# B&R Automation Studio project DuctLines (part 5)

#### Server.st - Cyclic code
```iecst
(********************************************************************
 ********************************************************************
 * Program: Server
 * File: Server.st
 * Created: May, 2018
 ********************************************************************
 * Implementation of program Server
 ********************************************************************)

PROGRAM _CYCLIC

	CASE Server.sStep OF

		0:  (* Open Ethernet Interface *)
			Server.TcpOpen_0.enable := 1;
			Server.TcpOpen_0.pIfAddr := 0;  (* Listen on all TCP/IP Interfaces*)
			Server.TcpOpen_0.port := 12000;  (* Port to listen*)
			Server.TcpOpen_0.options := 0;
			Server.TcpOpen_0;  (* Call the Function*)

			IF Server.TcpOpen_0.status = 0 THEN  (* TcpOpen successfull*)
				Server.sStep := 5;
			ELSIF Server.TcpOpen_0.status = ERR_FUB_BUSY THEN  (* TcpOpen not finished -> redo *)
				(* Busy *)
			ELSE  (* Goto Error Step *)
				Server.recv_timeout := 0;
				Server.sStep := 100;
			END_IF

		5:
			Server.linger_opt.lLinger := 0; (* linger Time = 0 *)
			Server.linger_opt.lOnOff := 1; (* linger Option ON *)
			Server.TcpIoctl_0.enable := 1;
			Server.TcpIoctl_0.ident := Server.TcpOpen_0.ident; (* Connection Ident from AsTCP.TCP_Open *)
			Server.TcpIoctl_0.ioctl := tcpSO_LINGER_SET; (* Set Linger Options *)
			Server.TcpIoctl_0.pData := ADR(Server.linger_opt);
			Server.TcpIoctl_0.datalen := SIZEOF(Server.linger_opt);
			Server.TcpIoctl_0;

			IF Server.TcpIoctl_0.status = 0 THEN  (* TcpIoctl successfull *)
				Server.sStep := 10;
			ELSIF Server.TcpIoctl_0.status = ERR_FUB_BUSY THEN  (* TcpIoctl not finished -> redo *)
				(* Busy *)
			ELSE  (* Goto Error Step *)
				Server.recv_timeout := 0;
				Server.sStep := 100;
			END_IF

		10: (* Wait for Client Connection *)
			Server.TcpServer_0.enable := 1;
			Server.TcpServer_0.ident := Server.TcpOpen_0.ident;  (* Connection Ident from AsTCP.TCP_Open *)
			Server.TcpServer_0.backlog := 1;  (* Number of clients waiting simultaneously for a connection*)
			Server.TcpServer_0.pIpAddr := ADR(Server.client_address);  (* Where to write the client IP-Address*)
			Server.TcpServer_0;  (* Call the Function*)

			IF Server.TcpServer_0.status = 0 THEN  (* Status = 0 if an client connects to server *)
				Server.sStep := 15;
			ELSIF Server.TcpServer_0.status = ERR_FUB_BUSY THEN  (* TcpServer not finished -> redo *)
				(* Busy *)
			ELSE  (* Goto Error Step *)
				Server.recv_timeout := 0;
				Server.sStep := 100;
			END_IF

		15:
			Server.TcpIoctl_0.enable := 1;
			Server.TcpIoctl_0.ident := Server.TcpServer_0.identclnt; (* Connection Ident from AsTCP.TCP_Server *)
			Server.TcpIoctl_0.ioctl := tcpSO_LINGER_SET;  (* Set Linger Options *)
			Server.TcpIoctl_0.pData := ADR(Server.linger_opt);
			Server.TcpIoctl_0.datalen := SIZEOF(Server.linger_opt);
			Server.TcpIoctl_0;

			IF Server.TcpIoctl_0.status = 0 THEN  (* TcpIoctl successfull *)
				Server.sStep := 20;
			ELSIF Server.TcpIoctl_0.status = ERR_FUB_BUSY THEN  (* TcpIoctl not finished -> redo *)
				(* Busy *)
			ELSE  (* Goto Error Step *)
				Server.recv_timeout := 0;
				Server.sStep := 100;
			END_IF

		20: (* Wait for Data *)
			Server.TcpRecv_0.enable := 1;
			Server.TcpRecv_0.ident := Server.TcpServer_0.identclnt;  (* Client Ident from AsTCP.TCP_Server *)
			Server.TcpRecv_0.pData	:= ADR(Server.data_buffer);  (* Where to store the incoming data *)
			Server.TcpRecv_0.datamax := SIZEOF(Server.data_buffer);  (* Length of data buffer *)
			Server.TcpRecv_0.flags := 0;
			Server.TcpRecv_0;  (* Call the Function*)

			IF Server.TcpRecv_0.status = 0 THEN
				(* This gets Server.sStep out of here when the PC program stop executing*)
				Server.recv_timeout := Server.recv_timeout + 1;
				IF Server.recv_timeout > 250 THEN
					Server.sStep := 40;
					Server.recv_timeout := 0;
				END_IF
			ELSIF Server.TcpRecv_0.status = tcpERR_NO_DATA THEN
				(*This criteria isn't true when the PC program isn't executing*)
				Server.recv_timeout := Server.recv_timeout + 1;
				IF Server.recv_timeout > 500 THEN
					Server.sStep := 40;
					Server.recv_timeout := 0;
				END_IF
			ELSIF Server.TcpRecv_0.status = ERR_FUB_BUSY THEN

			ELSIF Server.TcpRecv_0.status = tcpERR_NOT_CONNECTED THEN
				(* This doesn't appear to work.*)
				Server.sStep := 40;
			ELSE
				Server.recv_timeout := 0;
				Server.sStep := 100;
			END_IF

			LastByte := Server.TcpRecv_0.recvlen - 3;
			IF Server.data_buffer[LastByte] = 13 THEN
				(*Receive Transmission Complete, Parse Data*)
				Server.recv_timeout := 0;
				Server.data_buffer[LastByte] := 0;
				HandleIndex := 0;
				UpperLimit := LastByte; (* Parsing Loop Will Run To Here *)
				TrueString := 'True';
				Server.sStep := 25;
				(*Server.sStep := 90;*)
			END_IF
		25: (* Parse Out Values *)
			REPEAT
				(* Get The Tag Handle *)
				CommaPosition1 := HandleIndex;
				WHILE Server.data_buffer[CommaPosition1] <> 44 DO
					CommaPosition1 := CommaPosition1 + 1;
				END_WHILE;
				SLength := CommaPosition1 - HandleIndex;
				nxt_adr := memmove(ADR(HandleStringA), ADR(Server.data_buffer[HandleIndex]), SLength);
				HandleStringB := LEFT(HandleStringA, UDINT_TO_INT(SLength));
				TagHandle := atoi(ADR(HandleStringB));
				HandleIndex := CommaPosition1 + 1;

				(* Get The String Containing The Value *)
				CommaPosition1 := HandleIndex;
				WHILE Server.data_buffer[CommaPosition1] <> 44 DO
					CommaPosition1 := CommaPosition1 + 1;
				END_WHILE;
				SLength := CommaPosition1 - HandleIndex;
				nxt_adr := memmove(ADR(ValueStringA), ADR(Server.data_buffer[HandleIndex]), SLength);
				ValueStringB := LEFT(ValueStringA, UDINT_TO_INT(SLength));
				HandleIndex := CommaPosition1 + 1;
				CASE TagHandle OF
					0:
						RunJob := atoi(ADR(ValueStringB));
					1:
						IF strcmp(ADR(TrueString), ADR(ValueStringB)) = 0 THEN
							RunJobClick := TRUE;
						ELSE
							RunJobClick := FALSE;
						END_IF;
					2:
						NewRunJob := atoi(ADR(ValueStringB));
					3:
						IF strcmp(ADR(TrueString), ADR(ValueStringB)) = 0 THEN
							StartSignal := TRUE;
						ELSE
							StartSignal := FALSE;
						END_IF;
					4..9:
						ShearTable[TagHandle - 4] := atof(ADR(ValueStringB));
					10..15:
						LTNotchTable[TagHandle - 10] := atof(ADR(ValueStringB));
					16..21:
						VNotchTable[TagHandle - 16] := atof(ADR(ValueStringB));
					22..39:
						LeftHoleTable[TagHandle - 22] := atof(ADR(ValueStringB));
					40..57:
						CenterHoleTable[TagHandle - 40] := atof(ADR(ValueStringB));
					58..75:
						RightHoleTable[TagHandle - 58] := atof(ADR(ValueStringB));
					76:
						ShearHits := atoi(ADR(ValueStringB));
					77:
						LTNotchHits := atoi(ADR(ValueStringB));
					78:
						VNotchHits := atoi(ADR(ValueStringB));
					79:
						LeftHoleHits := atoi(ADR(ValueStringB));
					80:
						CenterHoleHits := atoi(ADR(ValueStringB));
					81:
						RightHoleHits := atoi(ADR(ValueStringB));
					82:
						IF strcmp(ADR(TrueString), ADR(ValueStringB)) = 0 THEN
							SealantRequired := TRUE;
						ELSE
							SealantRequired := FALSE;
						END_IF;
					83:
						IF strcmp(ADR(TrueString), ADR(ValueStringB)) = 0 THEN
							CropCut := TRUE;
						ELSE
							CropCut := FALSE;
						END_IF;
					84:
						WarningDelay1 := DINT_TO_TIME(atoi(ADR(ValueStringB)));
					85:
						PartsMade := atoi(ADR(ValueStringB));
					86:
						MetalDesired := atof(ADR(ValueStringB));
					87:
						MetalActual := atof(ADR(ValueStringB));
					88:
						IF strcmp(ADR(TrueString), ADR(ValueStringB)) = 0 THEN
							InCycle := TRUE;
						ELSE
							InCycle := FALSE;
						END_IF;
					89:
						PercentSpeed1 := atoi(ADR(ValueStringB));
					90:
						CropPercent1 := atoi(ADR(ValueStringB));
					91:
						TotalInches := atof(ADR(ValueStringB));
					92:
						PartLength := atof(ADR(ValueStringB));
					93:
					94:
						IF strcmp(ADR(TrueString), ADR(ValueStringB)) = 0 THEN
							MakeShearTable := TRUE;
						ELSE
							MakeShearTable := FALSE;
						END_IF;
					95:
						IF strcmp(ADR(TrueString), ADR(ValueStringB)) = 0 THEN
							MakeLTTable := TRUE;
						ELSE
							MakeLTTable := FALSE;
						END_IF;
					96:
						IF strcmp(ADR(TrueString), ADR(ValueStringB)) = 0 THEN
							MakeVTable := TRUE;
						ELSE
							MakeVTable := FALSE;
						END_IF;
					97:
						IF strcmp(ADR(TrueString), ADR(ValueStringB)) = 0 THEN
							MakeLHoleTable := TRUE;
						ELSE
							MakeLHoleTable := FALSE;
						END_IF;
					98:
						IF strcmp(ADR(TrueString), ADR(ValueStringB)) = 0 THEN
							MakeCHoleTable := TRUE;
						ELSE
							MakeCHoleTable := FALSE;
						END_IF;
					99:
						IF strcmp(ADR(TrueString), ADR(ValueStringB)) = 0 THEN
							MakeRHoleTable := TRUE;
						ELSE
							MakeRHoleTable := FALSE;
						END_IF;
					100:
						ShearFFlag := atoi(ADR(ValueStringB));
					101:
						NotchFFlag1 := atoi(ADR(ValueStringB));
					102:
						IF strcmp(ADR(TrueString), ADR(ValueStringB)) = 0 THEN
							BatchCancelSignal := TRUE;
						ELSE
							BatchCancelSignal := FALSE;
						END_IF;
					103:
						IF strcmp(ADR(TrueString), ADR(ValueStringB)) = 0 THEN
							RunContinuousSignal := TRUE;
						ELSE
							RunContinuousSignal := FALSE;
						END_IF;
					104:
						ShearJob := atoi(ADR(ValueStringB));
					105:
						LTJob := atoi(ADR(ValueStringB));
					106:
						VJob := atoi(ADR(ValueStringB));
					107:
						LHoleJob := atoi(ADR(ValueStringB));
					108:
					    BackGaugeJogPercent := atoi(ADR(ValueStringB)); (*Iowa Servo Brake Uses This, too*)
					109:
					    RHoleJob := atoi(ADR(ValueStringB)); (* Iowa *)
					    BackGaugeRunPercent := RHoleJob; (* Engel *)
					110:
						ShearDwell := atoi(ADR(ValueStringB));
					111:
						LTDwell := atoi(ADR(ValueStringB));
					112:
						VDwell := atoi(ADR(ValueStringB));
					113:
						LHoleDwell := atoi(ADR(ValueStringB));
					114:
						CHoleDwell := atoi(ADR(ValueStringB));
					115:
						RHoleDwell := atoi(ADR(ValueStringB));
					116:
						GapTime := atoi(ADR(ValueStringB));
					117..134:
						IF strcmp(ADR(TrueString), ADR(ValueStringB)) = 0 THEN
							LeftDiePosition[TagHandle - 117] := TRUE;
						ELSE
							LeftDiePosition[TagHandle - 117] := FALSE;
						END_IF;
					135..152:
						IF strcmp(ADR(TrueString), ADR(ValueStringB)) = 0 THEN
							CenterDiePosition[TagHandle - 135] := TRUE;
						ELSE
							CenterDiePosition[TagHandle - 135] := FALSE;
						END_IF;
					153..170:
						IF strcmp(ADR(TrueString), ADR(ValueStringB)) = 0 THEN
							RightDiePosition[TagHandle - 153] := TRUE;
						ELSE
							RightDiePosition[TagHandle - 153] := FALSE;
						END_IF;
					171:
						LTRemainder := atof(ADR(ValueStringB));
					172:
						VRemainder := atof(ADR(ValueStringB));
					173:
						LHoleRemainder := atof(ADR(ValueStringB));
					174:
						CHoleRemainder := atof(ADR(ValueStringB));
					175:
						RHoleRemainder := atof(ADR(ValueStringB));
					176:
						PercentJogSpeed1 := atoi(ADR(ValueStringB));
					177:
						MetalEncoder := atoi(ADR(ValueStringB));
					178:
						MarkEncoder := atoi(ADR(ValueStringB));
					179:
						PinspotEncoder := atoi(ADR(ValueStringB));
					180:
						BrakeEncoder := atoi(ADR(ValueStringB));
					181:
						IF strcmp(ADR(TrueString), ADR(ValueStringB)) = 0 THEN
							RollDriveEnableButton := TRUE;
						ELSE
							RollDriveEnableButton := FALSE;
						END_IF;
					182:
					(*Lift3DownDwell := STRING_TO_TIME(ValueStringB);*)
					    Lift3DownDwell := DINT_TO_TIME(atoi(ADR(ValueStringB)));
					183:
					(*Lift3UpDwell := STRING_TO_TIME(alueStringB);*)
					    Lift3UpDwell := DINT_TO_TIME(atoi(ADR(ValueStringB)));
					184:
						EngelBrakeModelNumber := atoi(ADR(ValueStringB));
					185:
						IF strcmp(ADR(TrueString), ADR(ValueStringB)) = 0 THEN
							SideDischargeBrake := TRUE;
						ELSE
							SideDischargeBrake := FALSE;
						END_IF;
					186: (* The E1000 PC program turns this on. *)
						IF strcmp(ADR(TrueString), ADR(ValueStringB)) = 0 THEN
							E1000CoilLine := TRUE;
						ELSE
							E1000CoilLine := FALSE;
						END_IF;
					187:
						BrakeEjectTarget := atof(ADR(ValueStringB));
					188..272: (*Obsolete Data*)
					273:
						LatestConnector := DINT_TO_INT(atoi(ADR(ValueStringB)));
					274:
						IF strcmp(ADR(TrueString), ADR(ValueStringB)) = 0 THEN
							WaitToFire1 := TRUE;
						ELSE
							WaitToFire1 := FALSE;
						END_IF;
					275:
						IF strcmp(ADR(TrueString), ADR(ValueStringB)) = 0 THEN
							WaitToFire2 := TRUE;
						ELSE
							WaitToFire2 := FALSE;
						END_IF;
					276:
						IF strcmp(ADR(TrueString), ADR(ValueStringB)) = 0 THEN
							WaitToFire3 := TRUE;
						ELSE
							WaitToFire3 := FALSE;
						END_IF;
					277: (*Obsolete Boolean*)
					278:
						MarkTableDecelDelay := atoi(ADR(ValueStringB));
					279:
						MarkGateUpDwell := atoi(ADR(ValueStringB));
					280:
						MarkPStartDelay := atoi(ADR(ValueStringB));
					281:
						MarkPPauseDwell := atoi(ADR(ValueStringB));
					282:
						MarkPStageTime := atoi(ADR(ValueStringB));
					283:
						MarkPStopDelay := atoi(ADR(ValueStringB));
					284:
						IF strcmp(ADR(TrueString), ADR(ValueStringB)) = 0 THEN
							BeginMarkHoming := TRUE;
						ELSE
							BeginMarkHoming := FALSE;
						END_IF;
					285:
						MarkTarget := atof(ADR(ValueStringB));
					286:
						MarkInPosBand := atoi(ADR(ValueStringB));
					287:
						MarkSlowBand := atoi(ADR(ValueStringB));
					288:
						MarkReference := atof(ADR(ValueStringB));
					289:
						MarkResolution := atof(ADR(ValueStringB));
					290:
						MarkStatus := atoi(ADR(ValueStringB));
					291:
						MarkMinLength := atof(ADR(ValueStringB));
					292:
						MarkDesired := atof(ADR(ValueStringB));
					293:
						MarkActual := atof(ADR(ValueStringB));
					294:
						IF strcmp(ADR(TrueString), ADR(ValueStringB)) = 0 THEN
							ClearLengthCountSignal := TRUE;
						ELSE
							ClearLengthCountSignal := FALSE;
						END_IF;
					295:
						IF strcmp(ADR(TrueString), ADR(ValueStringB)) = 0 THEN
							MarkButtonSignal := TRUE;
						ELSE
							MarkButtonSignal := FALSE;
						END_IF;
					296:
						IF strcmp(ADR(TrueString), ADR(ValueStringB)) = 0 THEN
							MarkSetSignal := TRUE;
						ELSE
							MarkSetSignal := FALSE;
						END_IF;
					297:
						TDCPushSetupDwell := atoi(ADR(ValueStringB));
					298:
						TDCSquareDelay := atoi(ADR(ValueStringB));
					299:
						TDCTablePauseDwell := atoi(ADR(ValueStringB));
					300:
						PinspotResolution := atof(ADR(ValueStringB));
					301:
						PSpotDesired := atof(ADR(ValueStringB));
					302:
						PSpotActual := atof(ADR(ValueStringB));
					303:
						IF strcmp(ADR(TrueString), ADR(ValueStringB)) = 0 THEN
							PinsRequired := TRUE;
						ELSE
							PinsRequired := FALSE;
						END_IF;
					304:
						PinTarget0 := atof(ADR(ValueStringB));
					305:
						PinTarget1 := atof(ADR(ValueStringB));
					306:
						PinTarget2 := atof(ADR(ValueStringB));
					307:
						PinTarget3 := atof(ADR(ValueStringB));
					308:
						PinTarget4 := atof(ADR(ValueStringB));
					309:
						PinTarget5 := atof(ADR(ValueStringB));
					310:
						PinTarget6 := atof(ADR(ValueStringB));
					311:
						PinTarget7 := atof(ADR(ValueStringB));
					312:
						PinTarget8 := atof(ADR(ValueStringB));
					313:
						PinTarget9 := atof(ADR(ValueStringB));
					314:
						PinRepeat0 := atoi(ADR(ValueStringB));
					315:
						PinRepeat1 := atoi(ADR(ValueStringB));
					316:
						PinRepeat2 := atoi(ADR(ValueStringB));
					317:
						PinRepeat3 := atoi(ADR(ValueStringB));
					318:
						PinRepeat4 := atoi(ADR(ValueStringB));
					319:
						PinRepeat5 := atoi(ADR(ValueStringB));
					320:
						PinRepeat6 := atoi(ADR(ValueStringB));
					321:
						PinRepeat7 := atoi(ADR(ValueStringB));
					322:
						PinRepeat8 := atoi(ADR(ValueStringB));
					323:
						PinRepeat9 := atoi(ADR(ValueStringB));
					324:
						PinDriveDwell := atoi(ADR(ValueStringB));
					325:
						PinLoadDwell := atoi(ADR(ValueStringB));
					326:
						PinLoadDelay := atoi(ADR(ValueStringB));
					327:
						IF strcmp(ADR(TrueString), ADR(ValueStringB)) = 0 THEN
							PinspotterSetSignal := TRUE;
						ELSE
							PinspotterSetSignal := FALSE;
						END_IF;
					328:
						IF strcmp(ADR(TrueString), ADR(ValueStringB)) = 0 THEN
							BrakeRefSignal := TRUE;
						ELSE
							BrakeRefSignal := FALSE;
						END_IF;
					329:
						BrakeReference := atof(ADR(ValueStringB));
					330:
						BrakeTarget0 := atof(ADR(ValueStringB));
					331:
						BrakeTarget1 := atof(ADR(ValueStringB));
					332:
						BrakeTarget2 := atof(ADR(ValueStringB));
					333:
						BrakeTarget3 := atof(ADR(ValueStringB));
					334:
						IF strcmp(ADR(TrueString), ADR(ValueStringB)) = 0 THEN
							BrakeRequired := TRUE;
						ELSE
							BrakeRequired := FALSE;
						END_IF;
					335:
						BrakeSlowWindow := atoi(ADR(ValueStringB)); (*Iowa*)
					    CoilLineSlowWindow := BrakeSlowWindow; (*Engel*)
					336:
						BrakeTargetWindow := atoi(ADR(ValueStringB)); (*Iowa*)
					    CoilLineTargetWindow := BrakeTargetWindow; (*Engel*)
					337:
						BrakeDesired := atof(ADR(ValueStringB));
					338:
						BrakeActual := atof(ADR(ValueStringB));
					339:
						BrakeResolution := atof(ADR(ValueStringB));
					340:
						DuctType := atoi(ADR(ValueStringB));
					341:
						BrakeStatus := atoi(ADR(ValueStringB));
					342:
						IF strcmp(ADR(TrueString), ADR(ValueStringB)) = 0 THEN
							PCBrakeSetSignal := TRUE;
						ELSE
							PCBrakeSetSignal := FALSE;
						END_IF;
					343:
						IF strcmp(ADR(TrueString), ADR(ValueStringB)) = 0 THEN
							FBBrakeSetSignal := TRUE;
						ELSE
							FBBrakeSetSignal := FALSE;
						END_IF;
					344:
						IF strcmp(ADR(TrueString), ADR(ValueStringB)) = 0 THEN
							ULineSelected := TRUE;
						ELSE
							ULineSelected := FALSE;
						END_IF;
					345:
						IF strcmp(ADR(TrueString), ADR(ValueStringB)) = 0 THEN
							ZeroCropCut := TRUE;
						ELSE
							ZeroCropCut := FALSE;
						END_IF;
					346:
						IF strcmp(ADR(TrueString), ADR(ValueStringB)) = 0 THEN
							Short2ndLeg := TRUE;
						ELSE
							Short2ndLeg := FALSE;
						END_IF;
					347:
						IF strcmp(ADR(TrueString), ADR(ValueStringB)) = 0 THEN
							HWBrakeWithPLC := TRUE;
						ELSE
							HWBrakeWithPLC := FALSE;
						END_IF;
					348:
						IF strcmp(ADR(TrueString), ADR(ValueStringB)) = 0 THEN
							LBrakeWithPLC := TRUE;
						ELSE
							LBrakeWithPLC := FALSE;
						END_IF;
					349:
						IF strcmp(ADR(TrueString), ADR(ValueStringB)) = 0 THEN
							CycleShear := TRUE;
						ELSE
							CycleShear := FALSE;
						END_IF;
					350:
						IF strcmp(ADR(TrueString), ADR(ValueStringB)) = 0 THEN
							CycleLTDie := TRUE;
						ELSE
							CycleLTDie := FALSE;
						END_IF;
					351:
						IF strcmp(ADR(TrueString), ADR(ValueStringB)) = 0 THEN
							CycleVDie := TRUE;
						ELSE
							CycleVDie := FALSE;
						END_IF;
					352:
						IF strcmp(ADR(TrueString), ADR(ValueStringB)) = 0 THEN
							CycleLDie := TRUE;
						ELSE
							CycleLDie := FALSE;
						END_IF;
					353:
						IF strcmp(ADR(TrueString), ADR(ValueStringB)) = 0 THEN
							CycleCDie := TRUE;
						ELSE
							CycleCDie := FALSE;
						END_IF;
					354:
						IF strcmp(ADR(TrueString), ADR(ValueStringB)) = 0 THEN
							CycleRDie := TRUE;
						ELSE
							CycleRDie := FALSE;
						END_IF;
					355:
						IF strcmp(ADR(TrueString), ADR(ValueStringB)) = 0 THEN
							SpareBool1 := TRUE;
						ELSE
							SpareBool1 := FALSE;
						END_IF;
					356:
						IF strcmp(ADR(TrueString), ADR(ValueStringB)) = 0 THEN
							ShearBrakeLatch := TRUE;
						ELSE
							ShearBrakeLatch := FALSE;
						END_IF;
					357:
						IF strcmp(ADR(TrueString), ADR(ValueStringB)) = 0 THEN
							CycleCustomVDie := TRUE;
						ELSE
							CycleCustomVDie := FALSE;
						END_IF;
					358:
						IF strcmp(ADR(TrueString), ADR(ValueStringB)) = 0 THEN
							CycleCustomLTDie := TRUE;
						ELSE
							CycleCustomLTDie := FALSE;
						END_IF;
					359:
						IF strcmp(ADR(TrueString), ADR(ValueStringB)) = 0 THEN
							SpareBool2 := TRUE;
						ELSE
							SpareBool2 := FALSE;
						END_IF;
					360:
						IF strcmp(ADR(TrueString), ADR(ValueStringB)) = 0 THEN
							SpareBool3 := TRUE;
						ELSE
							SpareBool3 := FALSE;
						END_IF;
					361:
						CustomLTDwell := atoi(ADR(ValueStringB));
					362:
						CustomVDwell := atoi(ADR(ValueStringB));
					363:
						TDCRFPusherStopDelay := atoi(ADR(ValueStringB));
					364:
						GlueApplicatorType := atoi(ADR(ValueStringB));
					365:
						IF strcmp(ADR(TrueString), ADR(ValueStringB)) = 0 THEN
							MakeButtonTable := TRUE;
						ELSE
							MakeButtonTable := FALSE;
						END_IF;
					366:
						IF strcmp(ADR(TrueString), ADR(ValueStringB)) = 0 THEN
							MakeShearBrakeTable := TRUE;
						ELSE
							MakeShearBrakeTable := FALSE;
						END_IF;
					367:
						IF strcmp(ADR(TrueString), ADR(ValueStringB)) = 0 THEN
							MakeCustomLTTable := TRUE;
						ELSE
							MakeCustomLTTable := FALSE;
						END_IF;
					368:
						IF strcmp(ADR(TrueString), ADR(ValueStringB)) = 0 THEN
							MakeCleatTable := TRUE;
						ELSE
							MakeCleatTable := FALSE;
						END_IF;
					369:
						ButtonHits := atoi(ADR(ValueStringB));
					370:
						ShearBrakeHits := atoi(ADR(ValueStringB));
					371:
						CustomLTHits := atoi(ADR(ValueStringB));
					372:
						CleatHits := atoi(ADR(ValueStringB));
					373:
						ButtonJob := atoi(ADR(ValueStringB));
					374:
						ShearBrakeJob := atoi(ADR(ValueStringB));
					375:
						CustomLTJob := atoi(ADR(ValueStringB));
					376:
						CleatJob := atoi(ADR(ValueStringB));
					377:
						ButtonRemainder := atof(ADR(ValueStringB));
					378:
						ShearBrakeRemainder := atof(ADR(ValueStringB));
					379:
						CustomLTRemainder := atof(ADR(ValueStringB));
					380:
						CleatRemainder := atof(ADR(ValueStringB));
					381..386:
						ButtonTable[TagHandle - 381] := atof(ADR(ValueStringB));
					387..392:
						ShearBrakeTable[TagHandle - 387] := atof(ADR(ValueStringB));
					393..398:
						CustomLTTable[TagHandle - 393] := atof(ADR(ValueStringB));
					399..404:
						CleatTable[TagHandle - 399] := atof(ADR(ValueStringB));
					405:
						DieUpDelay := atoi(ADR(ValueStringB));
					406:
						IF strcmp(ADR(TrueString), ADR(ValueStringB)) = 0 THEN
							BrakeAuto := TRUE;
						ELSE
							BrakeAuto := FALSE;
						END_IF;
					407:
						IF strcmp(ADR(TrueString), ADR(ValueStringB)) = 0 THEN
							DuctSelected := TRUE;
						ELSE
							DuctSelected := FALSE;
						END_IF;
					408:
						IF strcmp(ADR(TrueString), ADR(ValueStringB)) = 0 THEN
							EngelEServoOption := TRUE;
						ELSE
							EngelEServoOption := FALSE;
						END_IF;
					409:
						IF strcmp(ADR(TrueString), ADR(ValueStringB)) = 0 THEN
							ConfigureServos := TRUE;
						ELSE
							ConfigureServos := FALSE;
						END_IF;
					410:
						IF strcmp(ADR(TrueString), ADR(ValueStringB)) = 0 THEN
							SpareBool4 := TRUE;
						ELSE
							SpareBool4 := FALSE;
						END_IF;
					411:
						IF strcmp(ADR(TrueString), ADR(ValueStringB)) = 0 THEN
							SpareBool5 := TRUE;
						ELSE
							SpareBool5 := FALSE;
						END_IF;
					412:
						NotchFFlag2 := atoi(ADR(ValueStringB));
					413:
						ITmr1 := atoi(ADR(ValueStringB));
					414:
						ITmr2 := atoi(ADR(ValueStringB));
					415:
						ITmr3 := atoi(ADR(ValueStringB));
					416:
						ITmr4 := atoi(ADR(ValueStringB));
					417:
						ITmr5 := atoi(ADR(ValueStringB));
					418:
						ITmr6 := atoi(ADR(ValueStringB));
					419:
						ITmr7 := atoi(ADR(ValueStringB));
					420:
						ITmr8 := atoi(ADR(ValueStringB));
					421:
						ITmr9 := atoi(ADR(ValueStringB));
					422:
						ITmr10 := atoi(ADR(ValueStringB));
					423:
						ITmr11 := atoi(ADR(ValueStringB));
					424:
						ITmr12 := atoi(ADR(ValueStringB));
					425:
						ITmr13 := atoi(ADR(ValueStringB));
					426:
						IF strcmp(ADR(TrueString), ADR(ValueStringB)) = 0 THEN
							InsulationRequired := TRUE;
						ELSE
							InsulationRequired := FALSE;
						END_IF;
					427:
						IF strcmp(ADR(TrueString), ADR(ValueStringB)) = 0 THEN
							HeartBeat := TRUE;
						ELSE
							HeartBeat := FALSE;
						END_IF;
					428:
						IF strcmp(ADR(TrueString), ADR(ValueStringB)) = 0 THEN
							TDCRunSignal := TRUE;
						ELSE
							TDCRunSignal := FALSE;
						END_IF;
					429:
						IF strcmp(ADR(TrueString), ADR(ValueStringB)) = 0 THEN
							TDCRFMotor := TRUE;
						ELSE
							TDCRFMotor := FALSE;
						END_IF;
					430:
						IF strcmp(ADR(TrueString), ADR(ValueStringB)) = 0 THEN
							TDCPushSignal := TRUE;
						ELSE
							TDCPushSignal := FALSE;
						END_IF;
					431:
						IF strcmp(ADR(TrueString), ADR(ValueStringB)) = 0 THEN
							TDCPusherEnable := TRUE;
						ELSE
							TDCPusherEnable := FALSE;
						END_IF;
					432..481:
						IF strcmp(ADR(TrueString), ADR(ValueStringB)) = 0 THEN
							ButtonSignal[TagHandle - 432] := TRUE;
						ELSE
							ButtonSignal[TagHandle - 432] := FALSE;
						END_IF;
					482..531:
						IF strcmp(ADR(TrueString), ADR(ValueStringB)) = 0 THEN
							ButtonStatus[TagHandle - 482] := TRUE;
						ELSE
							ButtonStatus[TagHandle - 482] := FALSE;
						END_IF;
					532:
						IF strcmp(ADR(TrueString), ADR(ValueStringB)) = 0 THEN
							MarkRFInSignal := TRUE;
						ELSE
							MarkRFInSignal := FALSE;
						END_IF;
					533:
						IF strcmp(ADR(TrueString), ADR(ValueStringB)) = 0 THEN
							MarkRFOutSignal := TRUE;
						ELSE
							MarkRFOutSignal := FALSE;
						END_IF;
					534:
						IF strcmp(ADR(TrueString), ADR(ValueStringB)) = 0 THEN
							ExitBeltsOn := TRUE;
						ELSE
							ExitBeltsOn := FALSE;
						END_IF;
					535:
						IF strcmp(ADR(TrueString), ADR(ValueStringB)) = 0 THEN
							BrakeIsRefed := TRUE;
						ELSE
							BrakeIsRefed := FALSE;
						END_IF;
					536:
						IF strcmp(ADR(TrueString), ADR(ValueStringB)) = 0 THEN
							BrakeIsSetUp := TRUE;
						ELSE
							BrakeIsSetUp := FALSE;
						END_IF;
					537:
						WBPreset1 := DINT_TO_TIME(atoi(ADR(ValueStringB)));
					538:
						WBPreset2 := DINT_TO_TIME(atoi(ADR(ValueStringB)));
					539:
						WBPreset3 := DINT_TO_TIME(atoi(ADR(ValueStringB)));
					540:
						WBPreset4 := DINT_TO_TIME(atoi(ADR(ValueStringB)));
					541:
						WBPreset5 := DINT_TO_TIME(atoi(ADR(ValueStringB)));
					542:
						WBPreset6 := DINT_TO_TIME(atoi(ADR(ValueStringB)));
					543:
						MaleLeafDwell := atoi(ADR(ValueStringB));
					544:
						IF strcmp(ADR(TrueString), ADR(ValueStringB)) = 0 THEN
							PowerOn := TRUE;
						ELSE
							PowerOn := FALSE;
						END_IF;
					545:
						IF strcmp(ADR(TrueString), ADR(ValueStringB)) = 0 THEN
							TDCKnurlRollStyle := TRUE;
						ELSE
							TDCKnurlRollStyle := FALSE;
						END_IF;
					546:
						IF strcmp(ADR(TrueString), ADR(ValueStringB)) = 0 THEN
							TDCPusherStyle := TRUE;
						ELSE
							TDCPusherStyle := FALSE;
						END_IF;
					547:
						IF strcmp(ADR(TrueString), ADR(ValueStringB)) = 0 THEN
							ElectricWrapBrake := TRUE;
						ELSE
							ElectricWrapBrake := FALSE;
						END_IF;
					548:
						MetalGauge := atoi(ADR(ValueStringB));
					549:
						LightPGain := atoi(ADR(ValueStringB));
					550:
						MediumPGain := atoi(ADR(ValueStringB));
					551:
						HeavyPGain := atoi(ADR(ValueStringB));
					552:
						IF strcmp(ADR(TrueString), ADR(ValueStringB)) = 0 THEN
							DClampTest := TRUE;
						ELSE
							DClampTest := FALSE;
						END_IF;
					553:
						IF strcmp(ADR(TrueString), ADR(ValueStringB)) = 0 THEN
							UClampTest := TRUE;
						ELSE
							UClampTest := FALSE;
						END_IF;
					554:
						IF strcmp(ADR(TrueString), ADR(ValueStringB)) = 0 THEN
							DLeafTest := TRUE;
						ELSE
							DLeafTest := FALSE;
						END_IF;
					555:
						IF strcmp(ADR(TrueString), ADR(ValueStringB)) = 0 THEN
							ULeafTest := TRUE;
						ELSE
							ULeafTest := FALSE;
						END_IF;
					556:
						BDelay1 := atoi(ADR(ValueStringB));
					557:
						BDelay2 := atoi(ADR(ValueStringB));
					558:
						IF strcmp(ADR(TrueString), ADR(ValueStringB)) = 0 THEN
							ShearBrakeInstalled := TRUE;
						ELSE
							ShearBrakeInstalled := FALSE;
						END_IF;
					559:
						IF strcmp(ADR(TrueString), ADR(ValueStringB)) = 0 THEN
							PittsButton := TRUE;
						ELSE
							PittsButton := FALSE;
						END_IF;
					560:
						IF strcmp(ADR(TrueString), ADR(ValueStringB)) = 0 THEN
							PassThruButton := TRUE;
						ELSE
							PassThruButton := FALSE;
						END_IF;
					561:
						IF strcmp(ADR(TrueString), ADR(ValueStringB)) = 0 THEN
							SnapButton := TRUE;
						ELSE
							SnapButton := FALSE;
						END_IF;
					562:
						IF strcmp(ADR(TrueString), ADR(ValueStringB)) = 0 THEN
							PittsPosition := TRUE;
						ELSE
							PittsPosition := FALSE;
						END_IF;
					563:
						IF strcmp(ADR(TrueString), ADR(ValueStringB)) = 0 THEN
							PassThruPosition := TRUE;
						ELSE
							PassThruPosition := FALSE;
						END_IF;
					564:
						IF strcmp(ADR(TrueString), ADR(ValueStringB)) = 0 THEN
							SnapPosition := TRUE;
						ELSE
							SnapPosition := FALSE;
						END_IF;
					565:
						ColdSealLeadDelay := atoi(ADR(ValueStringB));
					566:
						ColdSealTrailDelay := atoi(ADR(ValueStringB));
					567:
						MarkTransferModel := atoi(ADR(ValueStringB));
					568:
						TDCTableLength := atof(ADR(ValueStringB));
					569:
						IF strcmp(ADR(TrueString), ADR(ValueStringB)) = 0 THEN
							LeftCleatEnable := TRUE;
						ELSE
							LeftCleatEnable := FALSE;
						END_IF;
					570:
						IF strcmp(ADR(TrueString), ADR(ValueStringB)) = 0 THEN
							RightCleatEnable := TRUE;
						ELSE
							RightCleatEnable := FALSE;
						END_IF;
					571:
						IF strcmp(ADR(TrueString), ADR(ValueStringB)) = 0 THEN
							InsulmaticSwingBlade := TRUE;
						ELSE
							InsulmaticSwingBlade := FALSE;
						END_IF;
					572:
						TDCRFPushDelay := atoi(ADR(ValueStringB));
					573:
						IF strcmp(ADR(TrueString), ADR(ValueStringB)) = 0 THEN
							BlockingValveButton := TRUE;
						ELSE
							BlockingValveButton := FALSE;
						END_IF;
					574:
						IF strcmp(ADR(TrueString), ADR(ValueStringB)) = 0 THEN
							MMCHeartBeat := TRUE;
						ELSE
							MMCHeartBeat := FALSE;
						END_IF;
					575:
						GlueLeadDelay := atoi(ADR(ValueStringB));
					576:
						GlueTrailDelay := atoi(ADR(ValueStringB));
					577:
						CleanCycleLength := atoi(ADR(ValueStringB));
					578:
						FlushTubeRaiseTime := atoi(ADR(ValueStringB));
					579:
						LightIGain := atoi(ADR(ValueStringB));
					580:
						MediumIGain := atoi(ADR(ValueStringB));
					581:
						HeavyIGain := atoi(ADR(ValueStringB));
					582:
						IF strcmp(ADR(TrueString), ADR(ValueStringB)) = 0 THEN
							GainsReceived := TRUE;
						ELSE
							GainsReceived := FALSE;
						END_IF;
					583:
						MaxSpeed1 := atof(ADR(ValueStringB));
					584:
						UnitsPerInch1 := atof(ADR(ValueStringB));
					585:
						AccelRampReal := atof(ADR(ValueStringB));
					586:
						DecelRampReal := atof(ADR(ValueStringB));
					587:
						BrakePGain := atoi(ADR(ValueStringB));
					588:
						BrakeIGain := atoi(ADR(ValueStringB));
					589:
						AccelRampReal2 := atof(ADR(ValueStringB));
					590:
						DecelRampReal2 := atof(ADR(ValueStringB));
					591:
						BrakePercentSpeed := atoi(ADR(ValueStringB));
					592:
						IF strcmp(ADR(TrueString), ADR(ValueStringB)) = 0 THEN
							ElectricDriveFaulted := TRUE;
						ELSE
							ElectricDriveFaulted := FALSE;
						END_IF;
					593:
						IF strcmp(ADR(TrueString), ADR(ValueStringB)) = 0 THEN
							InvertShuttle := TRUE;
						ELSE
							InvertShuttle := FALSE;
						END_IF;
					594:
						IF strcmp(ADR(TrueString), ADR(ValueStringB)) = 0 THEN
							HasInsulmaticOnInput := TRUE;
						ELSE
							HasInsulmaticOnInput := FALSE;
						END_IF;
					595:
						IF strcmp(ADR(TrueString), ADR(ValueStringB)) = 0 THEN
							StandAloneCleatRoller := TRUE;
						ELSE
							StandAloneCleatRoller := FALSE;
						END_IF;
					596:
						IF strcmp(ADR(TrueString), ADR(ValueStringB)) = 0 THEN
							MarkHeadJoggingIn := TRUE;
						ELSE
							MarkHeadJoggingIn := FALSE;
						END_IF;
					597:
						IF strcmp(ADR(TrueString), ADR(ValueStringB)) = 0 THEN
							MarkHeadJoggingOut := TRUE;
						ELSE
							MarkHeadJoggingOut := FALSE;
						END_IF;
					598:
						PivotTable := atoi(ADR(ValueStringB));
					599:
						KnurledRollLength := atof(ADR(ValueStringB));
					600:
						RotateCompleteLength := atof(ADR(ValueStringB));
					601:
						PivotClampLength := atof(ADR(ValueStringB));
					602..614:
						(*PivotTablePreset[TagHandle - 602] := atoi(ADR(ValueStringB));*)
					    PivotTablePreset[TagHandle - 602] := DINT_TO_TIME(atoi(ADR(ValueStringB)));
					615:
						CustomVMove := atof(ADR(ValueStringB));
					616:
						CustomVIndex := DINT_TO_USINT(atoi(ADR(ValueStringB)));
					617:
						IF strcmp(ADR(TrueString), ADR(ValueStringB)) = 0 THEN
							MakeCustomVTable := TRUE;
						ELSE
							MakeCustomVTable := FALSE;
						END_IF;
					618..623:
						CustomVTable[TagHandle - 618]:= atof(ADR(ValueStringB));
					624:
						CustomVHits := atoi(ADR(ValueStringB));
					625:
						CustomVJob := atoi(ADR(ValueStringB));
					626:
						CustomVRemainder := atof(ADR(ValueStringB));
					627:
						MarkCleanLength := atof(ADR(ValueStringB));
					628:
						MarkCleanDwell := atoi(ADR(ValueStringB));
					629:
						CleatControl := atoi(ADR(ValueStringB));
					630:
						CleatSide := atoi(ADR(ValueStringB));
					631:
						CleatOnDelay := atoi(ADR(ValueStringB));
					632:
						CleatOffDelay := atoi(ADR(ValueStringB));
					633:
						CoilWidth := atof(ADR(ValueStringB));
					634:
						IF strcmp(ADR(TrueString), ADR(ValueStringB)) = 0 THEN
							ZeroCropButton := TRUE;
						ELSE
							ZeroCropButton := FALSE;
						END_IF;
					635:
						ZeroCropOffset := atof(ADR(ValueStringB));
					636:
						IF strcmp(ADR(TrueString), ADR(ValueStringB)) = 0 THEN
							MakeBeadRollTable := TRUE;
						ELSE
							MakeBeadRollTable := FALSE;
						END_IF;
					637..646:
						BeadRollTable[TagHandle - 637] := atof(ADR(ValueStringB));
					647:
						BeadRollHits := atoi(ADR(ValueStringB));
					648:
						IF strcmp(ADR(TrueString), ADR(ValueStringB)) = 0 THEN
							ChangeBeadRoll := TRUE;
						ELSE
							ChangeBeadRoll := FALSE;
						END_IF;
					649:
						BeadRollJob := atoi(ADR(ValueStringB));
					650:
						IF strcmp(ADR(TrueString), ADR(ValueStringB)) = 0 THEN
							LBrakeWithNoPLC := TRUE;
						ELSE
							LBrakeWithNoPLC := FALSE;
						END_IF;
					651:
						IF strcmp(ADR(TrueString), ADR(ValueStringB)) = 0 THEN
							HWBrakeWithNoPLC := TRUE;
						ELSE
							HWBrakeWithNoPLC := FALSE;
						END_IF;
					652:
						IF strcmp(ADR(TrueString), ADR(ValueStringB)) = 0 THEN
							SlipAndDriveButton := TRUE;
						ELSE
							SlipAndDriveButton := FALSE;
						END_IF;
					653:
						IF strcmp(ADR(TrueString), ADR(ValueStringB)) = 0 THEN
							NotchShuttleValve := TRUE;
						ELSE
							NotchShuttleValve := FALSE;
						END_IF;
					654:
						IF strcmp(ADR(TrueString), ADR(ValueStringB)) = 0 THEN
							TDCNotchButton := TRUE;
						ELSE
							TDCNotchButton := FALSE;
						END_IF;
					655:
						FixedTDCHeadReference := atof(ADR(ValueStringB));
					656:
						FixedTDCHeadDesired := atof(ADR(ValueStringB));
					657:
						FixedTDCHeadActual := atof(ADR(ValueStringB));
					658:
						AdjustableTDCHeadReference := atof(ADR(ValueStringB));
					659:
						AdjustableTDCHeadDesired := atof(ADR(ValueStringB));
					660:
						AdjustableTDCHeadActual := atof(ADR(ValueStringB));
					661:
						TDCHomePosition := atof(ADR(ValueStringB));
					662:
						TDCHeadInPositionBand := atof(ADR(ValueStringB));
					663:
						TDCHeadSlowSpeedWindow := atof(ADR(ValueStringB));
					664:
						TDCHeadResolution := atof(ADR(ValueStringB));
					665:
						IF strcmp(ADR(TrueString), ADR(ValueStringB)) = 0 THEN
							TDCHeadReferenceButton := TRUE;
						ELSE
							TDCHeadReferenceButton := FALSE;
						END_IF;
					666:
						IF strcmp(ADR(TrueString), ADR(ValueStringB)) = 0 THEN
							TDCHeadReferenced := TRUE;
						ELSE
							TDCHeadReferenced := FALSE;
						END_IF;
					667:
						TDCFixedHeadPosition := atoi(ADR(ValueStringB));
					668:
						TDCAHeadPosition := atoi(ADR(ValueStringB));
					669:
						IF strcmp(ADR(TrueString), ADR(ValueStringB)) = 0 THEN
							TDCAutoWidthOption := TRUE;
						ELSE
							TDCAutoWidthOption := FALSE;
						END_IF;
					670:
						IF strcmp(ADR(TrueString), ADR(ValueStringB)) = 0 THEN
							TDCSetupOutputStyle := TRUE;
						ELSE
							TDCSetupOutputStyle := FALSE;
						END_IF;
					671:
						FittingDischargeType := atoi(ADR(ValueStringB));
					672..689:
						PunchSelect[TagHandle - 672] := atoi(ADR(ValueStringB));
					690:
						IF strcmp(ADR(TrueString), ADR(ValueStringB)) = 0 THEN
							HoleSize := TRUE;
						ELSE
							HoleSize := FALSE;
						END_IF;
					691:
						PunchMasterCoilWidth := atof(ADR(ValueStringB));
					692:
						IF strcmp(ADR(TrueString), ADR(ValueStringB)) = 0 THEN
							PunchMaster := TRUE;
						ELSE
							PunchMaster := FALSE;
						END_IF;
					693:
						IF strcmp(ADR(TrueString), ADR(ValueStringB)) = 0 THEN
							TDCTransferTableButton := TRUE;
						ELSE
							TDCTransferTableButton := FALSE;
						END_IF;
					694:
						IF strcmp(ADR(TrueString), ADR(ValueStringB)) = 0 THEN
							InsulmaticButton := TRUE;
						ELSE
							InsulmaticButton := FALSE;
						END_IF;
					695:
						IF strcmp(ADR(TrueString), ADR(ValueStringB)) = 0 THEN
							TDCTTLatch := TRUE;
						ELSE
							TDCTTLatch := FALSE;
						END_IF;
					696:
						IF strcmp(ADR(TrueString), ADR(ValueStringB)) = 0 THEN
							InsulmaticLatch := TRUE;
						ELSE
							InsulmaticLatch := FALSE;
						END_IF;
					697:
						IF strcmp(ADR(TrueString), ADR(ValueStringB)) = 0 THEN
							OneSpeedExitBelts := TRUE;
						ELSE
							OneSpeedExitBelts := FALSE;
						END_IF;
					1000: (*Update*)
						IF strcmp(ADR(TrueString), ADR(ValueStringB)) = 0 THEN
							UpdatePC := TRUE;
						ELSE
							UpdatePC := FALSE;
						END_IF;
				END_CASE;

				UNTIL
				HandleIndex >= UpperLimit
			END_REPEAT;
			Server.sStep := 20;
		30:	(* Send Data back to Client *)

			Server.TcpSend_0;  (* Call the Function*)

			IF Server.TcpSend_0.status = 0 THEN  (* Data sent *)
				Server.sStep := 20;	(* Go Wait For Another Transmission*)
			ELSIF Server.TcpSend_0.status = ERR_FUB_BUSY THEN  (* TcpSend not finished -> redo *)
				(* Busy *)
			ELSIF (Server.TcpSend_0.status = tcpERR_NOT_CONNECTED) THEN
				Server.sStep := 40;
			ELSE  (* Goto Error Step *)
				Server.recv_timeout := 0;
				Server.sStep := 100;
			END_IF

		40:
			Server.TcpClose_0.enable := 1;
			Server.TcpClose_0.ident := Server.TcpServer_0.identclnt;
			Server.TcpClose_0.how := 0;; // tcpSHUT_RD OR tcpSHUT_WR;
			Server.TcpClose_0;

			IF Server.TcpClose_0.status = 0 THEN
				Server.sStep := 50;
			ELSIF Server.TcpClose_0.status = ERR_FUB_BUSY THEN  (* TcpClose not finished -> redo *)
				(* Busy *)
			ELSE  (* Goto Error Step *)
				Server.recv_timeout := 0;
				Server.sStep := 100;
			END_IF
		50:
			Server.TcpClose_0.enable := 1;
			Server.TcpClose_0.ident := Server.TcpOpen_0.ident;
			Server.TcpClose_0.how := 0; //tcpSHUT_RD OR tcpSHUT_WR;
			Server.TcpClose_0;

			IF Server.TcpClose_0.status = 0 THEN
				Server.sStep := 0;
			ELSIF Server.TcpClose_0.status = ERR_FUB_BUSY THEN  (* TcpClose not finished -> redo *)
				(* Busy *)
			ELSE  (* Goto Error Step *)
				Server.recv_timeout := 0;
				Server.sStep := 100;
			END_IF

		100:  (* Here some error Handling has to be implemented *)
			Server.recv_timeout := Server.recv_timeout + 1;
			IF Server.recv_timeout > 250 THEN
				Server.sStep := 0; (* Try Again *)
            END_IF
	END_CASE

	IF Tracer < 32767 THEN
		Tracer := Tracer + 1;
	ELSE
		Tracer := 0;
	END_IF;

	IF UpdatePC THEN
		UpdatePC := FALSE;

        outStrLen := 0;
		outString := BOOL_TO_STRING(CropCut);
		itemStrLen := UINT_TO_UDINT(strlen(ADR(outString)));
		memcpy(ADR(Server.data_buffer[outStrLen]), ADR(outString), itemStrLen);
		outStrLen := outStrLen + itemStrLen;
		Server.data_buffer[outStrLen] := DINT_TO_BYTE(44); (*Comma*)
		outStrLen := outStrLen + 1;

		itoa(RunJob, ADR(outString));
		itemStrLen := UINT_TO_UDINT(strlen(ADR(outString)));
		memcpy(ADR(Server.data_buffer[outStrLen]), ADR(outString), itemStrLen);
		outStrLen := outStrLen + itemStrLen;
		Server.data_buffer[outStrLen] := DINT_TO_BYTE(44);
		outStrLen := outStrLen + 1;

		outString := BOOL_TO_STRING(StartSignal);
		itemStrLen := UINT_TO_UDINT(strlen(ADR(outString)));
		memcpy(ADR(Server.data_buffer[outStrLen]), ADR(outString), itemStrLen);
		outStrLen := outStrLen + itemStrLen;
		Server.data_buffer[outStrLen] := DINT_TO_BYTE(44);
		outStrLen := outStrLen + 1;

		outString := DINT_TO_STRING(PartsMade);
		itemStrLen := UINT_TO_UDINT(strlen(ADR(outString)));
		memcpy(ADR(Server.data_buffer[outStrLen]), ADR(outString), itemStrLen);
		outStrLen := outStrLen + itemStrLen;
		Server.data_buffer[outStrLen] := DINT_TO_BYTE(44);
		outStrLen := outStrLen + 1;

		outString := REAL_TO_STRING(TotalInches);
		itemStrLen := UINT_TO_UDINT(strlen(ADR(outString)));
		memcpy(ADR(Server.data_buffer[outStrLen]), ADR(outString), itemStrLen);
		outStrLen := outStrLen + itemStrLen;
		Server.data_buffer[outStrLen] := DINT_TO_BYTE(44);
		outStrLen := outStrLen + 1;

		outString := DINT_TO_STRING(MetalEncoder);
		itemStrLen := UINT_TO_UDINT(strlen(ADR(outString)));
		memcpy(ADR(Server.data_buffer[outStrLen]), ADR(outString), itemStrLen);
		outStrLen := outStrLen + itemStrLen;
		Server.data_buffer[outStrLen] := DINT_TO_BYTE(44);
		outStrLen := outStrLen + 1;

		outString := DINT_TO_STRING(MarkEncoder);
		itemStrLen := UINT_TO_UDINT(strlen(ADR(outString)));
		memcpy(ADR(Server.data_buffer[outStrLen]), ADR(outString), itemStrLen);
		outStrLen := outStrLen + itemStrLen;
		Server.data_buffer[outStrLen] := DINT_TO_BYTE(44);
		outStrLen := outStrLen + 1;

		outString := DINT_TO_STRING(PinspotEncoder);
		itemStrLen := UINT_TO_UDINT(strlen(ADR(outString)));
		memcpy(ADR(Server.data_buffer[outStrLen]), ADR(outString), itemStrLen);
		outStrLen := outStrLen + itemStrLen;
		Server.data_buffer[outStrLen] := DINT_TO_BYTE(44);
		outStrLen := outStrLen + 1;

		outString := REAL_TO_STRING(RealBrakePosition);
		itemStrLen := UINT_TO_UDINT(strlen(ADR(outString)));
		memcpy(ADR(Server.data_buffer[outStrLen]), ADR(outString), itemStrLen);
		outStrLen := outStrLen + itemStrLen;
		Server.data_buffer[outStrLen] := DINT_TO_BYTE(44);
		outStrLen := outStrLen + 1;

		outString := BOOL_TO_STRING(InCycle);
		itemStrLen := UINT_TO_UDINT(strlen(ADR(outString)));
		memcpy(ADR(Server.data_buffer[outStrLen]), ADR(outString), itemStrLen);
		outStrLen := outStrLen + itemStrLen;
		Server.data_buffer[outStrLen] := DINT_TO_BYTE(44);
		outStrLen := outStrLen + 1;

		outString := BOOL_TO_STRING(MakeShearTable);
		itemStrLen := UINT_TO_UDINT(strlen(ADR(outString)));
		memcpy(ADR(Server.data_buffer[outStrLen]), ADR(outString), itemStrLen);
		outStrLen := outStrLen + itemStrLen;
		Server.data_buffer[outStrLen] := DINT_TO_BYTE(44);
		outStrLen := outStrLen + 1;

		outString := BOOL_TO_STRING(MakeLTTable);
		itemStrLen := UINT_TO_UDINT(strlen(ADR(outString)));
		memcpy(ADR(Server.data_buffer[outStrLen]), ADR(outString), itemStrLen);
		outStrLen := outStrLen + itemStrLen;
		Server.data_buffer[outStrLen] := DINT_TO_BYTE(44);
		outStrLen := outStrLen + 1;

		outString := BOOL_TO_STRING(MakeVTable);
		itemStrLen := UINT_TO_UDINT(strlen(ADR(outString)));
		memcpy(ADR(Server.data_buffer[outStrLen]), ADR(outString), itemStrLen);
		outStrLen := outStrLen + itemStrLen;
		Server.data_buffer[outStrLen] := DINT_TO_BYTE(44);
		outStrLen := outStrLen + 1;

		outString := BOOL_TO_STRING(MakeLHoleTable);
		itemStrLen := UINT_TO_UDINT(strlen(ADR(outString)));
		memcpy(ADR(Server.data_buffer[outStrLen]), ADR(outString), itemStrLen);
		outStrLen := outStrLen + itemStrLen;
		Server.data_buffer[outStrLen] := DINT_TO_BYTE(44);
		outStrLen := outStrLen + 1;

		outString := BOOL_TO_STRING(MakeCHoleTable);
		itemStrLen := UINT_TO_UDINT(strlen(ADR(outString)));
		memcpy(ADR(Server.data_buffer[outStrLen]), ADR(outString), itemStrLen);
		outStrLen := outStrLen + itemStrLen;
		Server.data_buffer[outStrLen] := DINT_TO_BYTE(44);
		outStrLen := outStrLen + 1;

		outString := BOOL_TO_STRING(MakeRHoleTable);
		itemStrLen := UINT_TO_UDINT(strlen(ADR(outString)));
		memcpy(ADR(Server.data_buffer[outStrLen]), ADR(outString), itemStrLen);
		outStrLen := outStrLen + itemStrLen;
		Server.data_buffer[outStrLen] := DINT_TO_BYTE(44);
		outStrLen := outStrLen + 1;

		outString := BOOL_TO_STRING(ChangeConnector);
		itemStrLen := UINT_TO_UDINT(strlen(ADR(outString)));
		memcpy(ADR(Server.data_buffer[outStrLen]), ADR(outString), itemStrLen);
		outStrLen := outStrLen + itemStrLen;
		Server.data_buffer[outStrLen] := DINT_TO_BYTE(44);
		outStrLen := outStrLen + 1;

		outString := DINT_TO_STRING(MarkStatus);
		itemStrLen := UINT_TO_UDINT(strlen(ADR(outString)));
		memcpy(ADR(Server.data_buffer[outStrLen]), ADR(outString), itemStrLen);
		outStrLen := outStrLen + itemStrLen;
		Server.data_buffer[outStrLen] := DINT_TO_BYTE(44);
		outStrLen := outStrLen + 1;

		outString := BOOL_TO_STRING(MarkButtonSignal);
		itemStrLen := UINT_TO_UDINT(strlen(ADR(outString)));
		memcpy(ADR(Server.data_buffer[outStrLen]), ADR(outString), itemStrLen);
		outStrLen := outStrLen + itemStrLen;
		Server.data_buffer[outStrLen] := DINT_TO_BYTE(44);
		outStrLen := outStrLen + 1;

		outString := DINT_TO_STRING(BrakeStatus);
		itemStrLen := UINT_TO_UDINT(strlen(ADR(outString)));
		memcpy(ADR(Server.data_buffer[outStrLen]), ADR(outString), itemStrLen);
		outStrLen := outStrLen + itemStrLen;
		Server.data_buffer[outStrLen] := DINT_TO_BYTE(44);
		outStrLen := outStrLen + 1;

		outString := BOOL_TO_STRING(PCBrakeSetSignal);
		itemStrLen := UINT_TO_UDINT(strlen(ADR(outString)));
		memcpy(ADR(Server.data_buffer[outStrLen]), ADR(outString), itemStrLen);
		outStrLen := outStrLen + itemStrLen;
		Server.data_buffer[outStrLen] := DINT_TO_BYTE(44);
		outStrLen := outStrLen + 1;

		outString := BOOL_TO_STRING(MakeButtonTable);
		itemStrLen := UINT_TO_UDINT(strlen(ADR(outString)));
		memcpy(ADR(Server.data_buffer[outStrLen]), ADR(outString), itemStrLen);
		outStrLen := outStrLen + itemStrLen;
		Server.data_buffer[outStrLen] := DINT_TO_BYTE(44);
		outStrLen := outStrLen + 1;

		outString := BOOL_TO_STRING(MakeShearBrakeTable);
		itemStrLen := UINT_TO_UDINT(strlen(ADR(outString)));
		memcpy(ADR(Server.data_buffer[outStrLen]), ADR(outString), itemStrLen);
		outStrLen := outStrLen + itemStrLen;
		Server.data_buffer[outStrLen] := DINT_TO_BYTE(44);
		outStrLen := outStrLen + 1;

		outString := BOOL_TO_STRING(MakeCustomLTTable);
		itemStrLen := UINT_TO_UDINT(strlen(ADR(outString)));
		memcpy(ADR(Server.data_buffer[outStrLen]), ADR(outString), itemStrLen);
		outStrLen := outStrLen + itemStrLen;
		Server.data_buffer[outStrLen] := DINT_TO_BYTE(44);
		outStrLen := outStrLen + 1;

		outString := BOOL_TO_STRING(MakeCleatTable);
		itemStrLen := UINT_TO_UDINT(strlen(ADR(outString)));
		memcpy(ADR(Server.data_buffer[outStrLen]), ADR(outString), itemStrLen);
		outStrLen := outStrLen + itemStrLen;
		Server.data_buffer[outStrLen] := DINT_TO_BYTE(44);
		outStrLen := outStrLen + 1;

		outString := BOOL_TO_STRING(BrakeAuto);
		itemStrLen := UINT_TO_UDINT(strlen(ADR(outString)));
		memcpy(ADR(Server.data_buffer[outStrLen]), ADR(outString), itemStrLen);
		outStrLen := outStrLen + itemStrLen;
		Server.data_buffer[outStrLen] := DINT_TO_BYTE(44);
		outStrLen := outStrLen + 1;

		outString := BOOL_TO_STRING(DuctSelected);
		itemStrLen := UINT_TO_UDINT(strlen(ADR(outString)));
		memcpy(ADR(Server.data_buffer[outStrLen]), ADR(outString), itemStrLen);
		outStrLen := outStrLen + itemStrLen;
		Server.data_buffer[outStrLen] := DINT_TO_BYTE(44);
		outStrLen := outStrLen + 1;

		outString := BOOL_TO_STRING(TDCRFMotor);
		itemStrLen := UINT_TO_UDINT(strlen(ADR(outString)));
		memcpy(ADR(Server.data_buffer[outStrLen]), ADR(outString), itemStrLen);
		outStrLen := outStrLen + itemStrLen;
		Server.data_buffer[outStrLen] := DINT_TO_BYTE(44);
		outStrLen := outStrLen + 1;

		outString := BOOL_TO_STRING(TDCPusherEnable);
		itemStrLen := UINT_TO_UDINT(strlen(ADR(outString)));
		memcpy(ADR(Server.data_buffer[outStrLen]), ADR(outString), itemStrLen);
		outStrLen := outStrLen + itemStrLen;
		Server.data_buffer[outStrLen] := DINT_TO_BYTE(44);
		outStrLen := outStrLen + 1;

		outString := BOOL_TO_STRING(PowerOn);
		itemStrLen := UINT_TO_UDINT(strlen(ADR(outString)));
		memcpy(ADR(Server.data_buffer[outStrLen]), ADR(outString), itemStrLen);
		outStrLen := outStrLen + itemStrLen;
		Server.data_buffer[outStrLen] := DINT_TO_BYTE(44);
		outStrLen := outStrLen + 1;

		FOR Index := 0 TO 21 BY 1 DO
			outString := BOOL_TO_STRING(ButtonStatus[Index]);
			itemStrLen := UINT_TO_UDINT(strlen(ADR(outString)));
			memcpy(ADR(Server.data_buffer[outStrLen]), ADR(outString), itemStrLen);
			outStrLen := outStrLen + itemStrLen;
			Server.data_buffer[outStrLen] := DINT_TO_BYTE(44);
			outStrLen := outStrLen + 1;
  	    END_FOR;

		outString := BOOL_TO_STRING(PittsPosition);
		itemStrLen := UINT_TO_UDINT(strlen(ADR(outString)));
		memcpy(ADR(Server.data_buffer[outStrLen]), ADR(outString), itemStrLen);
		outStrLen := outStrLen + itemStrLen;
		Server.data_buffer[outStrLen] := DINT_TO_BYTE(44);
		outStrLen := outStrLen + 1;

		outString := BOOL_TO_STRING(PassThruPosition);
		itemStrLen := UINT_TO_UDINT(strlen(ADR(outString)));
		memcpy(ADR(Server.data_buffer[outStrLen]), ADR(outString), itemStrLen);
		outStrLen := outStrLen + itemStrLen;
		Server.data_buffer[outStrLen] := DINT_TO_BYTE(44);
		outStrLen := outStrLen + 1;

		outString := BOOL_TO_STRING(SnapPosition);
		itemStrLen := UINT_TO_UDINT(strlen(ADR(outString)));
		memcpy(ADR(Server.data_buffer[outStrLen]), ADR(outString), itemStrLen);
		outStrLen := outStrLen + itemStrLen;
		Server.data_buffer[outStrLen] := DINT_TO_BYTE(44);
		outStrLen := outStrLen + 1;

		outString := BOOL_TO_STRING(ElectricDriveFaulted);
		itemStrLen := UINT_TO_UDINT(strlen(ADR(outString)));
		memcpy(ADR(Server.data_buffer[outStrLen]), ADR(outString), itemStrLen);
		outStrLen := outStrLen + itemStrLen;
		Server.data_buffer[outStrLen] := DINT_TO_BYTE(44);
		outStrLen := outStrLen + 1;

		outString := BOOL_TO_STRING(MarkRFInSignal);
		itemStrLen := UINT_TO_UDINT(strlen(ADR(outString)));
		memcpy(ADR(Server.data_buffer[outStrLen]), ADR(outString), itemStrLen);
		outStrLen := outStrLen + itemStrLen;
		Server.data_buffer[outStrLen] := DINT_TO_BYTE(44);
		outStrLen := outStrLen + 1;

		outString := BOOL_TO_STRING(MarkRFOutSignal);
		itemStrLen := UINT_TO_UDINT(strlen(ADR(outString)));
		memcpy(ADR(Server.data_buffer[outStrLen]), ADR(outString), itemStrLen);
		outStrLen := outStrLen + itemStrLen;
		Server.data_buffer[outStrLen] := DINT_TO_BYTE(44);
		outStrLen := outStrLen + 1;

		outString := BOOL_TO_STRING(MakeCustomVTable);
		itemStrLen := UINT_TO_UDINT(strlen(ADR(outString)));
		memcpy(ADR(Server.data_buffer[outStrLen]), ADR(outString), itemStrLen);
		outStrLen := outStrLen + itemStrLen;
		Server.data_buffer[outStrLen] := DINT_TO_BYTE(44);
		outStrLen := outStrLen + 1;

		outString := BOOL_TO_STRING(ZeroCropCut);
		itemStrLen := UINT_TO_UDINT(strlen(ADR(outString)));
		memcpy(ADR(Server.data_buffer[outStrLen]), ADR(outString), itemStrLen);
		outStrLen := outStrLen + itemStrLen;
		Server.data_buffer[outStrLen] := DINT_TO_BYTE(44);
		outStrLen := outStrLen + 1;

		outString := DINT_TO_STRING(BeadRollHits);
		itemStrLen := UINT_TO_UDINT(strlen(ADR(outString)));
		memcpy(ADR(Server.data_buffer[outStrLen]), ADR(outString), itemStrLen);
		outStrLen := outStrLen + itemStrLen;
		Server.data_buffer[outStrLen] := DINT_TO_BYTE(44);
		outStrLen := outStrLen + 1;

		outString := BOOL_TO_STRING(MakeBeadRollTable);
		itemStrLen := UINT_TO_UDINT(strlen(ADR(outString)));
		memcpy(ADR(Server.data_buffer[outStrLen]), ADR(outString), itemStrLen);
		outStrLen := outStrLen + itemStrLen;
		Server.data_buffer[outStrLen] := DINT_TO_BYTE(44);
		outStrLen := outStrLen + 1;

		outString := BOOL_TO_STRING(ChangeBeadRoll);
		itemStrLen := UINT_TO_UDINT(strlen(ADR(outString)));
		memcpy(ADR(Server.data_buffer[outStrLen]), ADR(outString), itemStrLen);
		outStrLen := outStrLen + itemStrLen;
		Server.data_buffer[outStrLen] := DINT_TO_BYTE(44);
		outStrLen := outStrLen + 1;

		outString := BOOL_TO_STRING(NotchShuttleValve);
		itemStrLen := UINT_TO_UDINT(strlen(ADR(outString)));
		memcpy(ADR(Server.data_buffer[outStrLen]), ADR(outString), itemStrLen);
		outStrLen := outStrLen + itemStrLen;
		Server.data_buffer[outStrLen] := DINT_TO_BYTE(44);
		outStrLen := outStrLen + 1;

		outString := BOOL_TO_STRING(TDCHeadReferenced);
		itemStrLen := UINT_TO_UDINT(strlen(ADR(outString)));
		memcpy(ADR(Server.data_buffer[outStrLen]), ADR(outString), itemStrLen);
		outStrLen := outStrLen + itemStrLen;
		Server.data_buffer[outStrLen] := DINT_TO_BYTE(44);
		outStrLen := outStrLen + 1;

		outString := DINT_TO_STRING(TDCFixedHeadPosition);
		itemStrLen := UINT_TO_UDINT(strlen(ADR(outString)));
		memcpy(ADR(Server.data_buffer[outStrLen]), ADR(outString), itemStrLen);
		outStrLen := outStrLen + itemStrLen;
		Server.data_buffer[outStrLen] := DINT_TO_BYTE(44);
		outStrLen := outStrLen + 1;

		outString := DINT_TO_STRING(TDCAHeadPosition);
		itemStrLen := UINT_TO_UDINT(strlen(ADR(outString)));
		memcpy(ADR(Server.data_buffer[outStrLen]), ADR(outString), itemStrLen);
		outStrLen := outStrLen + itemStrLen;
		Server.data_buffer[outStrLen] := DINT_TO_BYTE(44);
		outStrLen := outStrLen + 1;

		outString := BOOL_TO_STRING(TDCTTLatch);
		itemStrLen := UINT_TO_UDINT(strlen(ADR(outString)));
		memcpy(ADR(Server.data_buffer[outStrLen]), ADR(outString), itemStrLen);
		outStrLen := outStrLen + itemStrLen;
		Server.data_buffer[outStrLen] := DINT_TO_BYTE(44);
		outStrLen := outStrLen + 1;

		outString := BOOL_TO_STRING(InsulmaticLatch);
		itemStrLen := UINT_TO_UDINT(strlen(ADR(outString)));
		memcpy(ADR(Server.data_buffer[outStrLen]), ADR(outString), itemStrLen);
		outStrLen := outStrLen + itemStrLen;
		Server.data_buffer[outStrLen] := DINT_TO_BYTE(44);
		outStrLen := outStrLen + 1;

		(*Add end of transmission signal*)
		Server.data_buffer[outStrLen] := DINT_TO_BYTE(13);
		outStrLen := outStrLen + 1;

		(*Setup and make 1st call to Server.TcpSend_0*)
		Server.TcpSend_0.enable := 1;
		Server.TcpSend_0.ident := Server.TcpServer_0.identclnt;  (* Client Ident from AsTCP.TCP_Server *)
		Server.TcpSend_0.pData := ADR(Server.data_buffer);  (* Which data to send *)
		Server.TcpSend_0.datalen := outStrLen;  (* Length of data to send *)
		Server.TcpSend_0.flags := 0;
		Server.TcpSend_0;  (* Call the Function*)
		Server.sStep := 30;
	END_IF;

END_PROGRAM
```

#### Server.typ - TCP Server Variables
```iecst
(********************************************************************
 * COPYRIGHT -- Bernecker + Rainer
 ********************************************************************
 * Package: LibAsTCP
 * File: LibAsTCP.typ
 * Author: Bernecker + Rainer
 * Created: February 21, 2008
 ********************************************************************
 * Data types of package LibAsTCP
 ********************************************************************)

TYPE
	Server_typ : 	STRUCT  (*TCP Server Variables*)
		sStep : UINT; (*TCP Server Step Variable*)
		client_address : STRING[20]; (*Address of the client connection to the Server*)
		TcpOpen_0 : TcpOpen; (*AsTCP.TcpOpen FUB*)
		TcpServer_0 : TcpServer; (*AsTCP.TcpServer FUB*)
		TcpRecv_0 : TcpRecv; (*AsTCP.TcpRecv FUB*)
		TcpSend_0 : TcpSend; (*AsTCP.TcpSend FUB*)
		TcpClose_0 : TcpClose; (*AsTCP.TcpClose FUB*)
		TcpIoctl_0 : TcpIoctl; (*AsTCP.TcpIoctl*)
		data_buffer : ARRAY[0..4096]OF BYTE; (*Data buffer ( receive and send )*)
		linger_opt : tcpLINGER_typ; (*AsTCP.tcpLINGER_typ*)
		recv_timeout : UDINT; (*receive timeout*)
	END_STRUCT;
END_TYPE
```

#### Server.var - Data for Server Task
```iecst
(********************************************************************
 * COPYRIGHT -- Bernecker + Rainer
 ********************************************************************
 * Package: LibAsTCP
 * File: LibAsTCP.var
 * Author: Bernecker + Rainer
 * Created: February 21, 2008
 ********************************************************************
 * Variables of package LibAsTCP
 ********************************************************************)
VAR
	itemStrLen : UDINT;
	outStrLen : UDINT;
	outString : STRING[80];
	UpdatePC : BOOL;
	CommaPosition1 : UDINT;
	HandleIndex : UDINT;
	HandleStringA : STRING[80];
	HandleStringB : STRING[80];
	LastByte : UDINT;
	nxt_adr : UDINT;
	Server : Server_typ := (0); (*Data for Server Task*)
	SLength : UDINT;
	TagHandle : DINT;
	Tracer : DINT;
	Index : DINT;
	TrueString : STRING[80];
	UpperLimit : UDINT;
	ValueStringA : STRING[80];
	ValueStringB : STRING[80];
END_VAR
```

### Program Logical/LibAsTCP1_ST/Client (IEC) - AsTCP Client Application

#### Client.st - Cyclic code
```iecst
(********************************************************************
 * COPYRIGHT -- Bernecker + Rainer
 ********************************************************************
 * Program: Client
 * File: Client.st
 * Author: Bernecker + Rainer
 * Created: February 21, 2008
 ********************************************************************
 * Implementation of program Client
 ********************************************************************)

PROGRAM _CYCLIC

	(*LibAsTCP1_ST.send_data[0] := LibAsTCP1_ST.send_data[0] + 1; *) (* Generate a "running" variable for Data transfer*)
	testDINT := 63;
	Client.sStep := 100;

	CASE Client.sStep OF

		 0: (* Open Ethernet Interface *)
			Client.TcpOpen_0.enable := 1;
			Client.TcpOpen_0.pIfAddr := 0;  (* Which Interface to open *)
			Client.TcpOpen_0.port := 12001;  (* Port on client side to use *)
			Client.TcpOpen_0.options := 0;
			Client.TcpOpen_0;  (* Call the Function *)

			IF Client.TcpOpen_0.status = 0 THEN  (* TcpOpen successfull *)
				Client.sStep := 5;
			ELSIF Client.TcpOpen_0.status = ERR_FUB_BUSY THEN  (* TcpOpen not finished -> redo *)
			  (* Busy *)
			ELSE  (* Goto Error Step *)
				Client.sStep := 100;
			END_IF

		 5:
		 	Client.linger_opt.lLinger := 0; (* linger Time = 0 *)
			Client.linger_opt.lOnOff := 1; (* linger Option ON *)

		 	Client.TcpIoctl_0.enable := 1;
			Client.TcpIoctl_0.ident := Client.TcpOpen_0.ident; (* Connection Ident from AsTP.TCP_Open *)
			Client.TcpIoctl_0.ioctl := tcpSO_LINGER_SET; (* Set Linger Options *)
			Client.TcpIoctl_0.pData := ADR(Client.linger_opt);
			Client.TcpIoctl_0.datalen := SIZEOF(Client.linger_opt);
   			Client.TcpIoctl_0;

			IF Client.TcpIoctl_0.status = 0 THEN  (* TcpIoctl successfull *)
				Client.sStep := 10;
			ELSIF Client.TcpIoctl_0.status = ERR_FUB_BUSY THEN  (* TcpIoctl not finished -> redo *)
			  (* Busy *)
			ELSE  (* Goto Error Step *)
				Client.sStep := 100;
			END_IF

		10: (* Connect to the other Station *)
			Client.TcpClient_0.enable := 1;
			Client.TcpClient_0.ident := Client.TcpOpen_0.ident;  (* Connection Ident from AsTCP.TCP_Open *)
			Client.TcpClient_0.portserv := 12002;  (* Port on server side to use *)
			(*Client.TcpClient_0.pServer := ADR('10.43.28.115');*)  (* Server Address *)
			Client.TcpClient_0.pServer := ADR('127.0.0.2');
			Client.TcpClient_0;  (* Call the Function*)

			IF Client.TcpClient_0.status = 0 THEN  (* Open ok -> Send Data *)
				Client.sStep := 20;
			ELSIF Client.TcpClient_0.status = ERR_FUB_BUSY THEN  (* TcpClient not finished -> redo *)
			  (* Busy *)
			ELSIF Client.TcpClient_0.status = tcpERR_INVALID THEN  (* Port error -> Close actual connection, and reopen a new one *)
				Client.sStep := 40;
			ELSE  (* Goto Error Step *)
				Client.sStep := 100;
			END_IF

		20: (* Send Data to the Server *)
			Client.TcpSend_0.enable := 1;
			Client.TcpSend_0.ident := Client.TcpOpen_0.ident;  (* Connection Ident from AsTCP.TCP_Open *)
			Client.TcpSend_0.pData := ADR(LibAsTCP1_ST.send_data);  (* Which data to send *)
			(*Client.TcpSend_0.datalen := SIZEOF(LibAsTCP1_ST.send_data);*)  (* Length of data to send *)
			Client.TcpSend_0.datalen := 4;
			Client.TcpSend_0.flags := 0;
			Client.TcpSend_0;  (* Call the Function*)

			IF Client.TcpSend_0.status = 0 THEN  (* Data was sent sucessfully -> receive data *)
				Client.sStep := 30;
			ELSIF Client.TcpSend_0.status = ERR_FUB_BUSY THEN  (* TcpSend not finished -> redo *)
			  (* Busy *)
			ELSIF (Client.TcpSend_0.status = tcpERR_SENTLEN) OR (Client.TcpSend_0.status = tcpERR_NOT_CONNECTED) THEN (* Connection Lost *)
				Client.sStep := 40;
			ELSE  (* Goto Error Step *)
				Client.sStep := 100;
			END_IF

	    30: (* Receive Data from the Server *)
			Client.TcpRecv_0.enable := 1;
			Client.TcpRecv_0.ident := Client.TcpOpen_0.ident; (* Connection Ident from AsTCP.TCP_Open *)
			Client.TcpRecv_0.pData	:= ADR(LibAsTCP1_ST.receive_data);  (* Where to store the incoming data *)
			Client.TcpRecv_0.datamax := SIZEOF(LibAsTCP1_ST.receive_data);  (* Lenght of data buffer *)
			Client.TcpRecv_0.flags := 0;
			Client.TcpRecv_0;  (* Call the Function*)

			IF Client.TcpRecv_0.status = 0 THEN  (* Data was received sucessfully -> Send next packet *)
				(*Client.sStep := 20;*)
				Client.sStep := 50;
				BytesReceived := Client.TcpRecv_0.recvlen;
				Client.recv_timeout := 0;
			ELSIF Client.TcpRecv_0.status = tcpERR_NO_DATA THEN  (* No data received - wait *)
			  Client.recv_timeout := Client.recv_timeout + 1;
			  IF Client.recv_timeout > 500 THEN
					(*Client.sStep := 40;*)
					Client.sStep := 55;
				Client.recv_timeout := 0;
			  END_IF
			  (* No Data received *)
			ELSIF Client.TcpRecv_0.status = ERR_FUB_BUSY THEN  (* TcpRecv not finished -> redo *)
			  (* Busy *)
			ELSIF Client.TcpRecv_0.status = tcpERR_NOT_CONNECTED THEN (* Connection Lost *)
				(*Client.sStep := 40;*)
				Client.sStep := 60;
			ELSE  (* Goto Error Step *)
				Client.sStep := 100;
			END_IF

		40: (* Close connection *)
			Client.TcpClose_0.enable := 1;
			Client.TcpClose_0.ident := Client.TcpOpen_0.ident;  (* Connection Ident from AsTCP.TCP_Open *)
			Client.TcpClose_0.how := 0;
			Client.TcpClose_0;  (* Call the Function*)

			IF Client.TcpClose_0.status = 0 THEN  (* Close sucessfull -> Reopen the interface *)
				Client.sStep := 0;
			ELSIF Client.TcpClose_0.status = ERR_FUB_BUSY THEN  (* TcpClose not finished -> redo *)
			  (* Busy *)
			ELSE  (* Goto Error Step *)
				Client.sStep := 100;
			END_IF

	   100: (* Here some error Handling has to be implemented *)

	END_CASE

END_PROGRAM
```

#### Client.var - Data for Client Task
```iecst
(********************************************************************
 * COPYRIGHT -- Bernecker + Rainer
 ********************************************************************
 * Package: LibAsTCP
 * File: LibAsTCP.var
 * Author: Bernecker + Rainer
 * Created: February 21, 2008
 ********************************************************************
 * Variables of package LibAsTCP
 ********************************************************************)
VAR
	testDINT : DINT;
	testString : STRING[80];
	Tracer : USINT;
	BytesReceived : UDINT;
	Client : Client_typ := (0); (*Data for Client Task*)
END_VAR
```

- Library Logical/LibAsTCP1_ST/Library (IEC) (no source held here)

### Program Logical/MarkTable (IEC)

#### Variables.var
```iecst
VAR
	BackUpParts : BOOL;
	DirectionDelay : BOOL;
	ForwardDelay : TIME;
	Gate2 : BOOL;
	Gate3 : BOOL;
	GateLowerDelay : TIME;
	GateReset : BOOL;
	GateUpTime : TIME;
	MarkPusherStopDOB : BOOL;
	PSettled : BOOL;
	Psh1 : BOOL;
	Psh2 : BOOL;
	Psh3 : BOOL;
	Psh4 : BOOL;
	Psh5 : BOOL;
	Psh6 : BOOL;
	Psh8 : BOOL;
	Psh9 : BOOL;
	Psh10 : BOOL;
	Psh11 : BOOL;
	PshPauseTmrDone : BOOL;
	PshStageTmrDone : BOOL;
	PshStartTmrDone : BOOL;
	PshStopDelayTmrDone : BOOL;
	PusherOffDelay : TIME;
	PushReverse : BOOL;
	PushValve2 : BOOL;
	PushValve3 : BOOL;
	ReverseDelay : TIME;
	SettleTime : TIME;
	SetupPushers : {REDUND_UNREPLICABLE} BOOL := FALSE;
	Step1 : BOOL;
	Step2 : BOOL;
	Step3 : BOOL;
	Step4 : BOOL;
	Step5 : BOOL;
	Step6 : BOOL;
	Step7 : BOOL;
	Step8 : BOOL;
	Step9 : BOOL;
	Step11 : BOOL;
	Step12 : BOOL;
	Step13 : BOOL;
	Step14 : BOOL;
	Step15 : BOOL;
	TableFwd2 : BOOL;
	TableFwd3 : BOOL;
	TableRev2 : BOOL;
	TableRev3 : BOOL;
	TableStyle2 : BOOL;
	TableStyle3 : BOOL;
	tmDirectionDelay : TIME;
	tmMPS : TIME;
	tmMPSD : TIME;
	tmMPSDelay : TIME;
	tmPPDwell : TIME;
	TOF_0 : TOF;
	TOF_1 : TOF;
	TON_0 : TON;
	TON_1 : TON;
	TON_2 : TON;
	TON_3 : TON;
	TON_4 : TON;
	TON_5 : TON;
	TON_6 : TON;
	TON_7 : TON;
	TON_8 : TON;
	TON_9 : TON;
	TON_10 : TON;
	truepart : BOOL;
	truepartoff : BOOL;
	WaitDone : BOOL;
	TON_11 : TON;
	TON_12 : TON;
	ReverfseDelay : TIME;
	MarkTableLatch : BOOL;
	TON_13 : TON;
	MarkPushReady : BOOL;
	MPRTime : TIME;
	TOF_2 : TOF;
	Step6A : BOOL;
	Step13A : BOOL;
END_VAR
```

#### Cyclic.ld
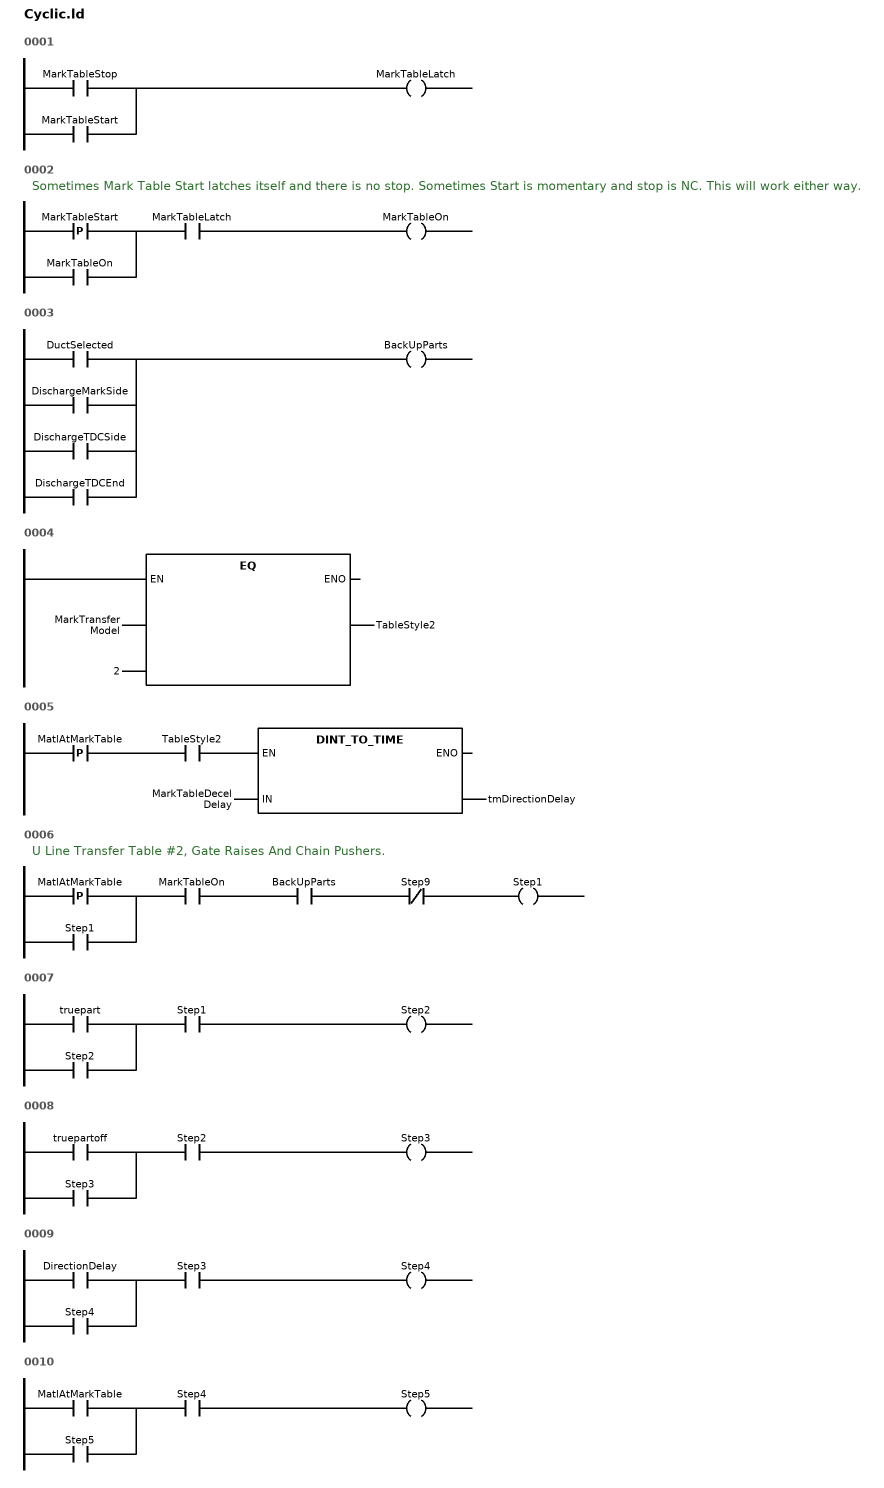
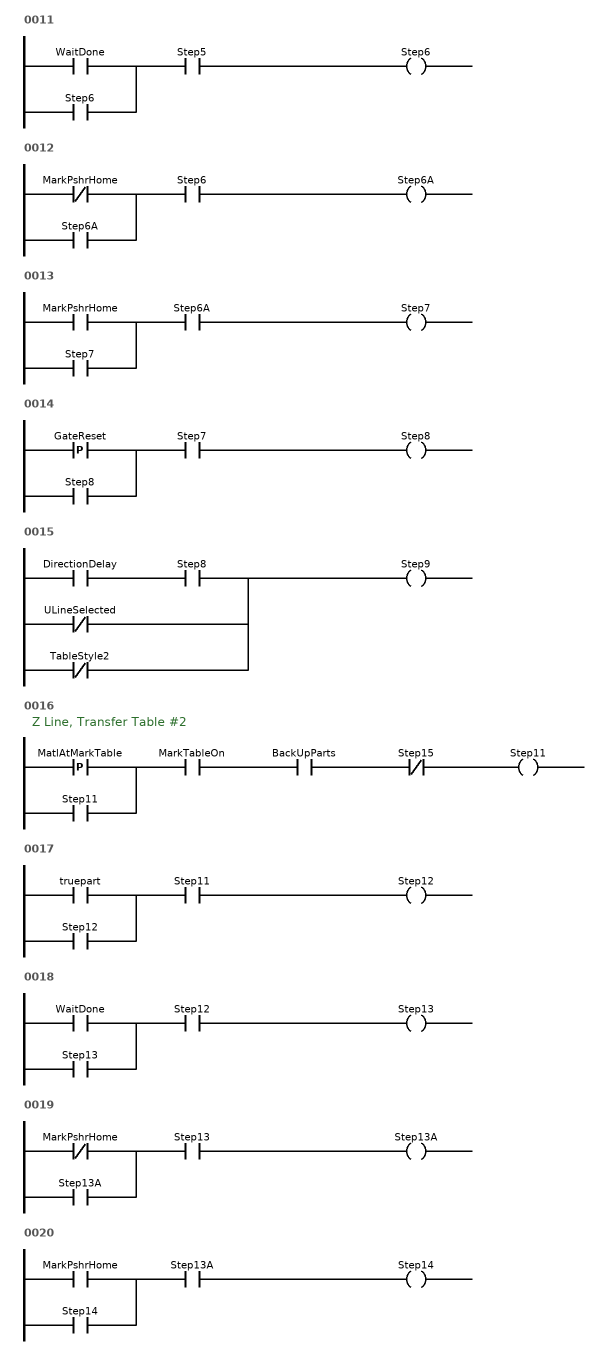
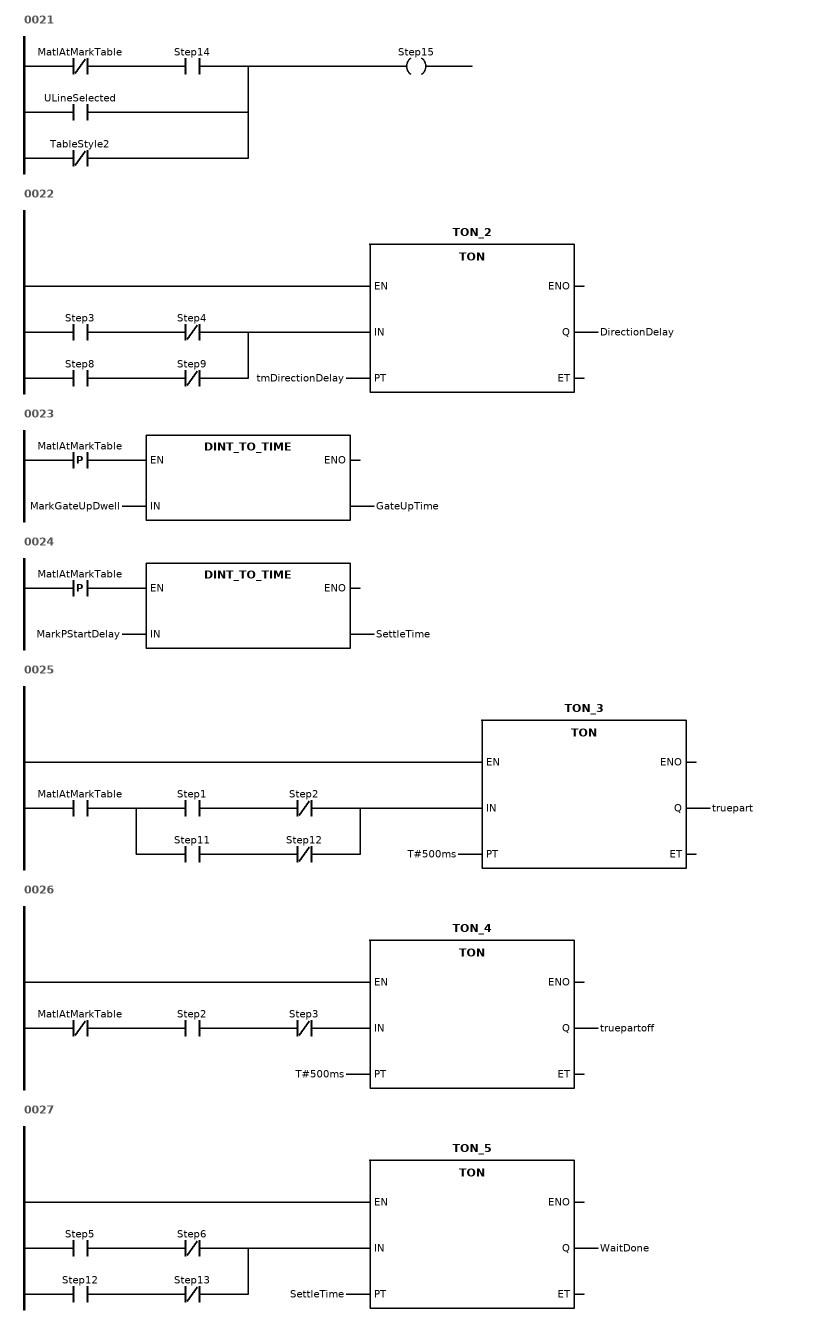
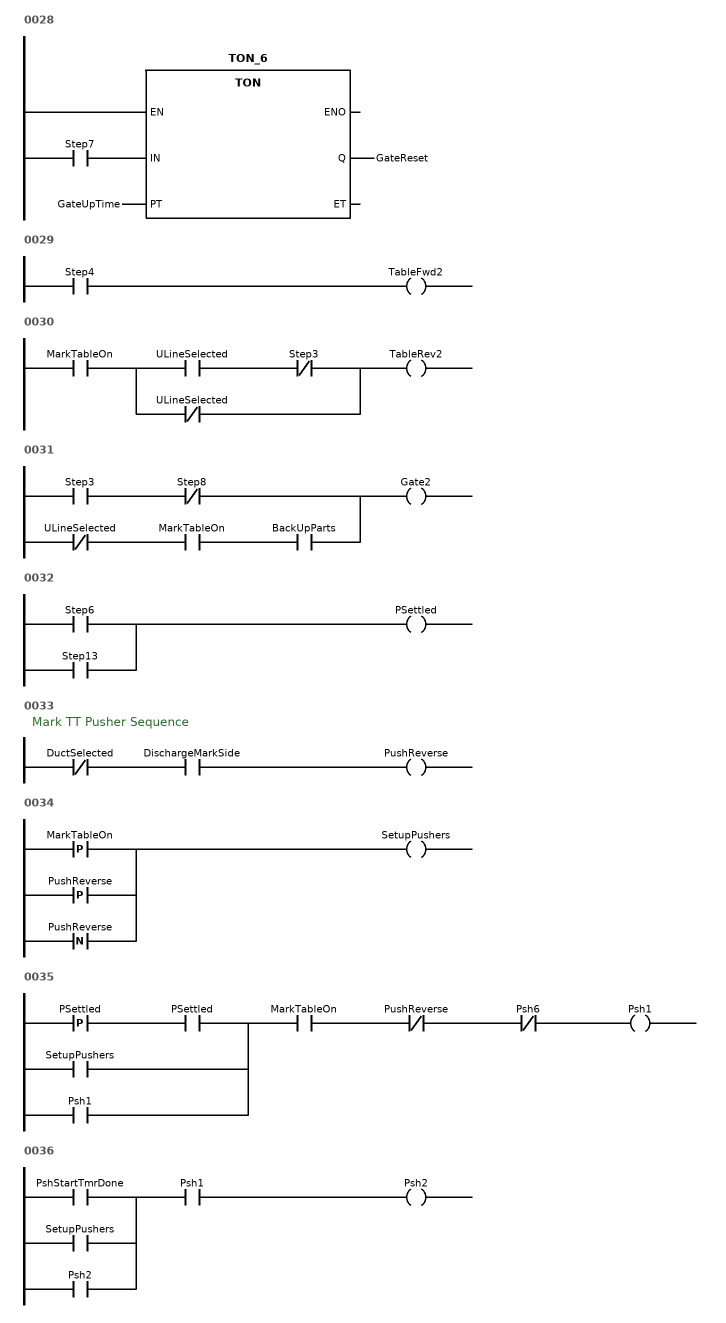
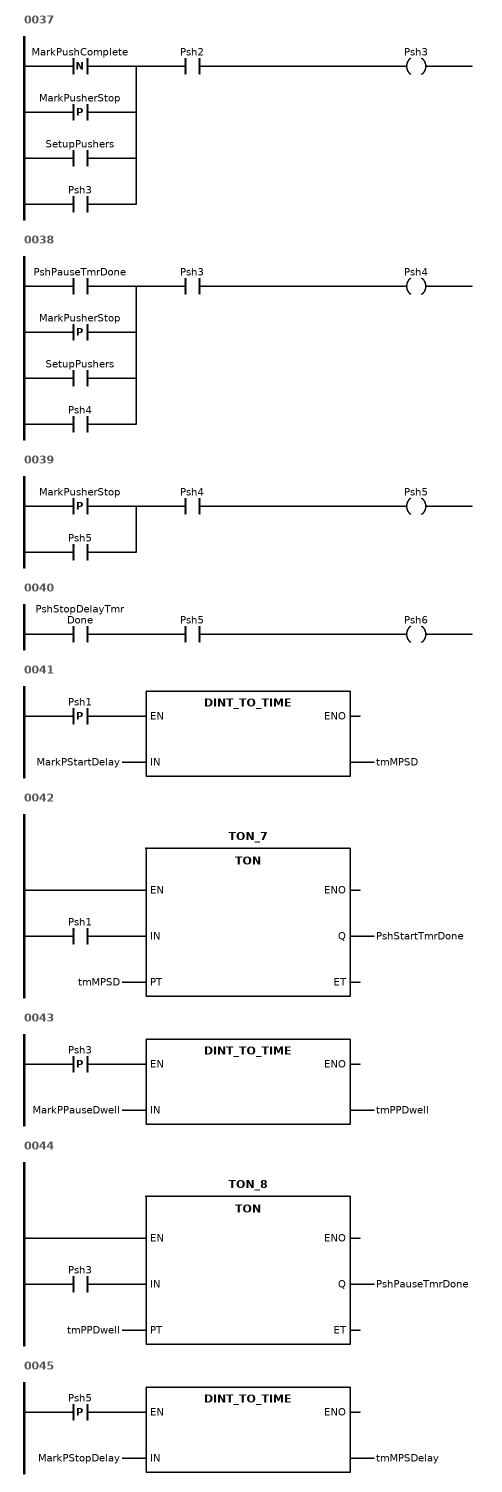
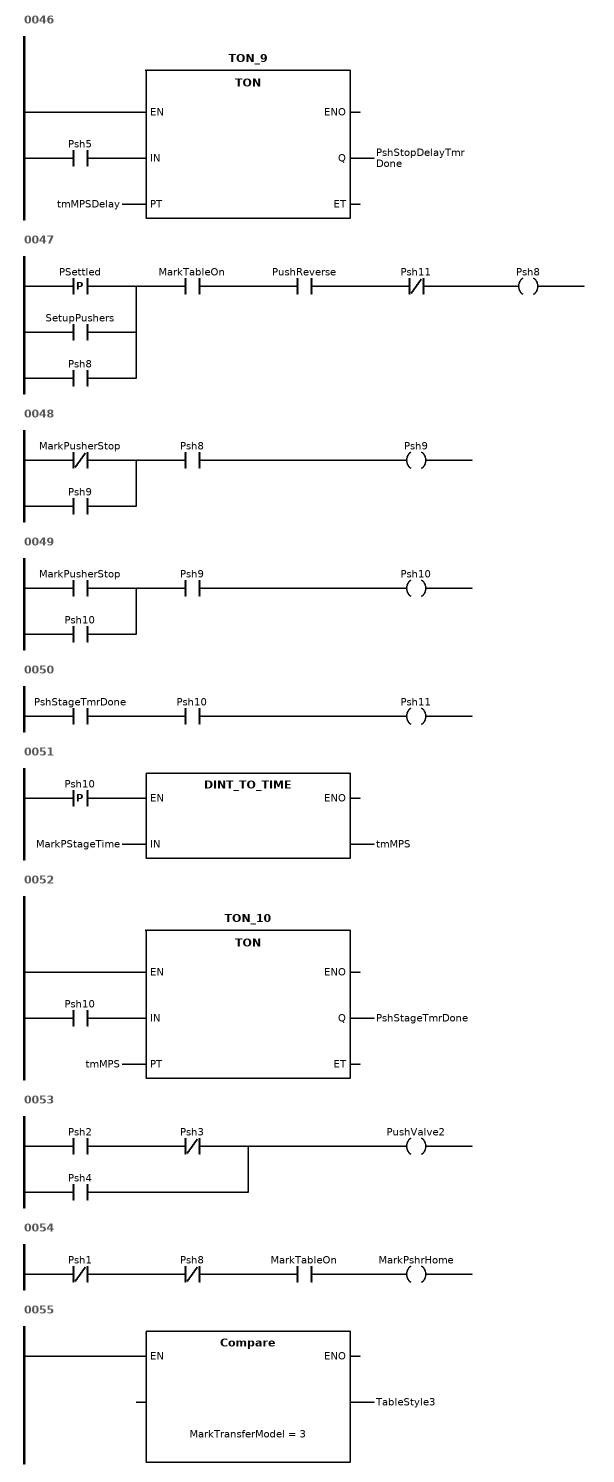
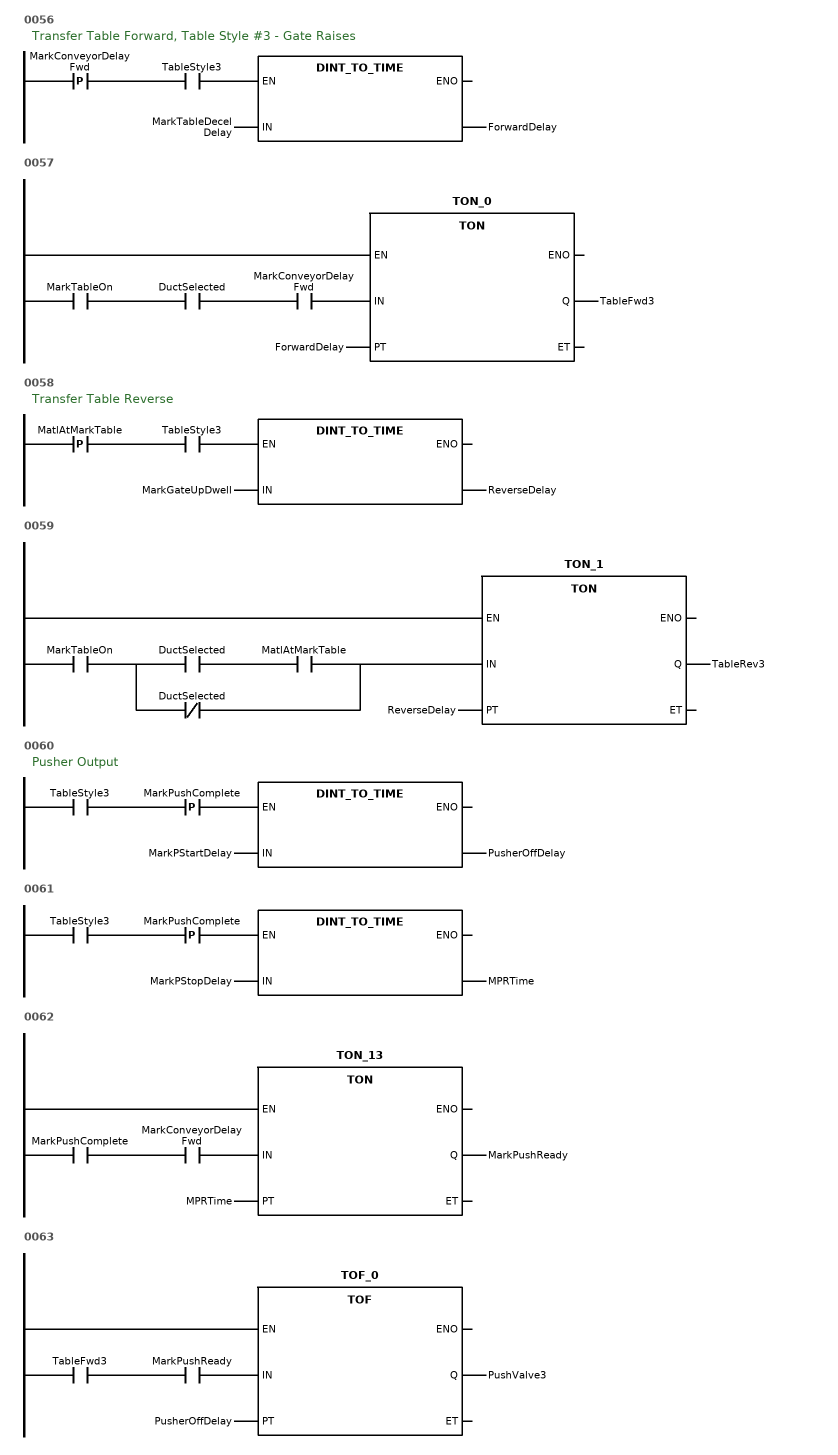
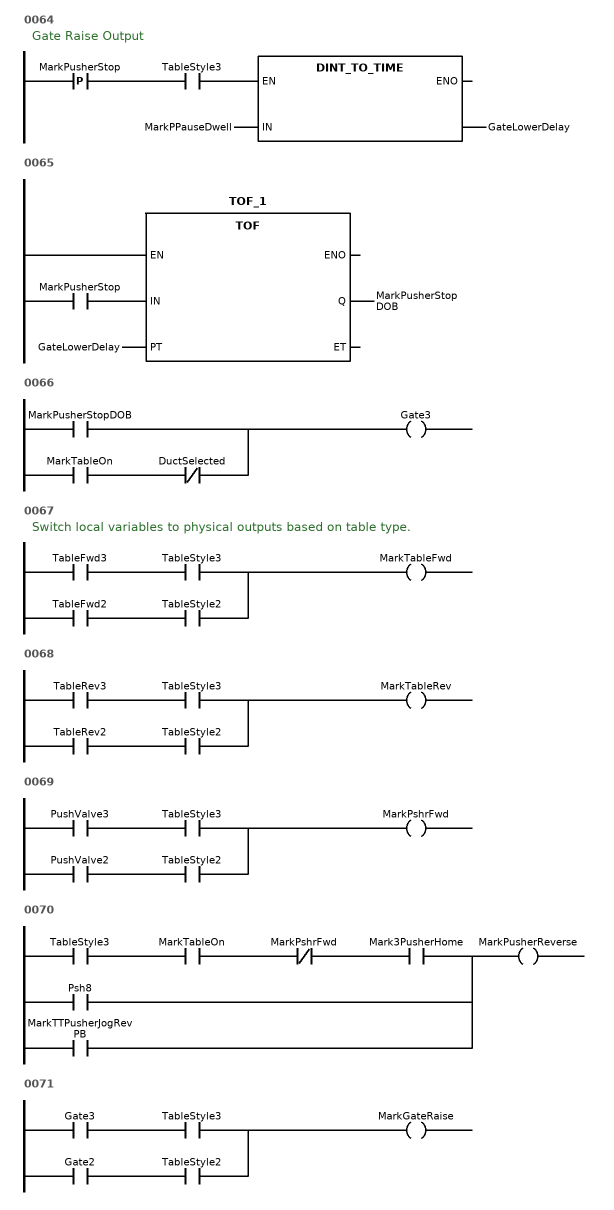
Ladder, written as Structured Text:
```iecst
PROGRAM _CYCLIC
VAR
    _e1 : R_TRIG;
    _e2 : R_TRIG;
    _e3 : R_TRIG;
    _e4 : R_TRIG;
    _e5 : R_TRIG;
    _e6 : R_TRIG;
    _e7 : R_TRIG;
    _e8 : R_TRIG;
    _e9 : R_TRIG;
    _e10 : F_TRIG;
    _e11 : R_TRIG;
    _e12 : F_TRIG;
    _e13 : R_TRIG;
    _e14 : R_TRIG;
    _e15 : R_TRIG;
    _e16 : R_TRIG;
    _e17 : R_TRIG;
    _e18 : R_TRIG;
    _e19 : R_TRIG;
    _e20 : R_TRIG;
    _e21 : R_TRIG;
    _e22 : R_TRIG;
    _e23 : R_TRIG;
    _e24 : R_TRIG;
    _e25 : R_TRIG;
END_VAR
(* Network 1 *)
MarkTableLatch := MarkTableStop OR MarkTableStart;

(* Network 2: Sometimes Mark Table Start latches itself and there is no stop. Sometimes Start is momentary and stop is NC. This will work either way. *)
_e1(CLK := MarkTableStart);
MarkTableOn := (_e1.Q OR MarkTableOn) AND MarkTableLatch;

(* Network 3 *)
BackUpParts := DuctSelected OR DischargeMarkSide OR DischargeTDCSide OR DischargeTDCEnd;

(* Network 4 *)
TableStyle2 := MarkTransferModel = 2;

(* Network 5 *)
_e2(CLK := MatlAtMarkTable);
IF _e2.Q AND TableStyle2 THEN tmDirectionDelay := DINT_TO_TIME(MarkTableDecelDelay); END_IF;

(* Network 6: U Line Transfer Table #2, Gate Raises And Chain Pushers. *)
_e3(CLK := MatlAtMarkTable);
Step1 := (_e3.Q OR Step1) AND MarkTableOn AND BackUpParts AND NOT Step9;

(* Network 7 *)
Step2 := (truepart OR Step2) AND Step1;

(* Network 8 *)
Step3 := (truepartoff OR Step3) AND Step2;

(* Network 9 *)
Step4 := (DirectionDelay OR Step4) AND Step3;

(* Network 10 *)
Step5 := (MatlAtMarkTable OR Step5) AND Step4;

(* Network 11 *)
Step6 := (WaitDone OR Step6) AND Step5;

(* Network 12 *)
Step6A := (NOT MarkPshrHome OR Step6A) AND Step6;

(* Network 13 *)
Step7 := (MarkPshrHome OR Step7) AND Step6A;

(* Network 14 *)
_e4(CLK := GateReset);
Step8 := (_e4.Q OR Step8) AND Step7;

(* Network 15 *)
Step9 := (DirectionDelay AND Step8) OR NOT ULineSelected OR NOT TableStyle2;

(* Network 16: Z Line, Transfer Table #2 *)
_e5(CLK := MatlAtMarkTable);
Step11 := (_e5.Q OR Step11) AND MarkTableOn AND BackUpParts AND NOT Step15;

(* Network 17 *)
Step12 := (truepart OR Step12) AND Step11;

(* Network 18 *)
Step13 := (WaitDone OR Step13) AND Step12;

(* Network 19 *)
Step13A := (NOT MarkPshrHome OR Step13A) AND Step13;

(* Network 20 *)
Step14 := (MarkPshrHome OR Step14) AND Step13A;

(* Network 21 *)
Step15 := (NOT MatlAtMarkTable AND Step14) OR ULineSelected OR NOT TableStyle2;

(* Network 22 *)
TON_2(IN := (Step3 AND NOT Step4) OR (Step8 AND NOT Step9), PT := tmDirectionDelay);
DirectionDelay := TON_2.Q;

(* Network 23 *)
_e6(CLK := MatlAtMarkTable);
IF _e6.Q THEN GateUpTime := DINT_TO_TIME(MarkGateUpDwell); END_IF;

(* Network 24 *)
_e7(CLK := MatlAtMarkTable);
IF _e7.Q THEN SettleTime := DINT_TO_TIME(MarkPStartDelay); END_IF;

(* Network 25 *)
TON_3(IN := MatlAtMarkTable AND ((Step1 AND NOT Step2) OR (Step11 AND NOT Step12)), PT := T#500ms);
truepart := TON_3.Q;

(* Network 26 *)
TON_4(IN := NOT MatlAtMarkTable AND Step2 AND NOT Step3, PT := T#500ms);
truepartoff := TON_4.Q;

(* Network 27 *)
TON_5(IN := (Step5 AND NOT Step6) OR (Step12 AND NOT Step13), PT := SettleTime);
WaitDone := TON_5.Q;

(* Network 28 *)
TON_6(IN := Step7, PT := GateUpTime);
GateReset := TON_6.Q;

(* Network 29 *)
TableFwd2 := Step4;

(* Network 30 *)
TableRev2 := MarkTableOn AND ((ULineSelected AND NOT Step3) OR NOT ULineSelected);

(* Network 31 *)
Gate2 := (Step3 AND NOT Step8) OR (NOT ULineSelected AND MarkTableOn AND BackUpParts);

(* Network 32 *)
PSettled := Step6 OR Step13;

(* Network 33: Mark TT Pusher Sequence *)
PushReverse := NOT DuctSelected AND DischargeMarkSide;

(* Network 34 *)
_e8(CLK := MarkTableOn);
_e9(CLK := PushReverse);
_e10(CLK := PushReverse);
SetupPushers := _e8.Q OR _e9.Q OR _e10.Q;

(* Network 35 *)
_e11(CLK := PSettled);
Psh1 := ((_e11.Q AND PSettled) OR SetupPushers OR Psh1) AND MarkTableOn AND NOT PushReverse AND NOT Psh6;

(* Network 36 *)
Psh2 := (PshStartTmrDone OR SetupPushers OR Psh2) AND Psh1;

(* Network 37 *)
_e12(CLK := MarkPushComplete);
_e13(CLK := MarkPusherStop);
Psh3 := (_e12.Q OR _e13.Q OR SetupPushers OR Psh3) AND Psh2;

(* Network 38 *)
_e14(CLK := MarkPusherStop);
Psh4 := (PshPauseTmrDone OR _e14.Q OR SetupPushers OR Psh4) AND Psh3;

(* Network 39 *)
_e15(CLK := MarkPusherStop);
Psh5 := (_e15.Q OR Psh5) AND Psh4;

(* Network 40 *)
Psh6 := PshStopDelayTmrDone AND Psh5;

(* Network 41 *)
_e16(CLK := Psh1);
IF _e16.Q THEN tmMPSD := DINT_TO_TIME(MarkPStartDelay); END_IF;

(* Network 42 *)
TON_7(IN := Psh1, PT := tmMPSD);
PshStartTmrDone := TON_7.Q;

(* Network 43 *)
_e17(CLK := Psh3);
IF _e17.Q THEN tmPPDwell := DINT_TO_TIME(MarkPPauseDwell); END_IF;

(* Network 44 *)
TON_8(IN := Psh3, PT := tmPPDwell);
PshPauseTmrDone := TON_8.Q;

(* Network 45 *)
_e18(CLK := Psh5);
IF _e18.Q THEN tmMPSDelay := DINT_TO_TIME(MarkPStopDelay); END_IF;

(* Network 46 *)
TON_9(IN := Psh5, PT := tmMPSDelay);
PshStopDelayTmrDone := TON_9.Q;

(* Network 47 *)
_e19(CLK := PSettled);
Psh8 := (_e19.Q OR SetupPushers OR Psh8) AND MarkTableOn AND PushReverse AND NOT Psh11;

(* Network 48 *)
Psh9 := (NOT MarkPusherStop OR Psh9) AND Psh8;

(* Network 49 *)
Psh10 := (MarkPusherStop OR Psh10) AND Psh9;

(* Network 50 *)
Psh11 := PshStageTmrDone AND Psh10;

(* Network 51 *)
_e20(CLK := Psh10);
IF _e20.Q THEN tmMPS := DINT_TO_TIME(MarkPStageTime); END_IF;

(* Network 52 *)
TON_10(IN := Psh10, PT := tmMPS);
PshStageTmrDone := TON_10.Q;

(* Network 53 *)
PushValve2 := (Psh2 AND NOT Psh3) OR Psh4;

(* Network 54 *)
MarkPshrHome := NOT Psh1 AND NOT Psh8 AND MarkTableOn;

(* Network 55 *)
TableStyle3 := MarkTransferModel = 3;

(* Network 56: Transfer Table Forward, Table Style #3 - Gate Raises *)
_e21(CLK := MarkConveyorDelayFwd);
IF _e21.Q AND TableStyle3 THEN ForwardDelay := DINT_TO_TIME(MarkTableDecelDelay); END_IF;

(* Network 57 *)
TON_0(IN := MarkTableOn AND DuctSelected AND MarkConveyorDelayFwd, PT := ForwardDelay);
TableFwd3 := TON_0.Q;

(* Network 58: Transfer Table Reverse *)
_e22(CLK := MatlAtMarkTable);
IF _e22.Q AND TableStyle3 THEN ReverseDelay := DINT_TO_TIME(MarkGateUpDwell); END_IF;

(* Network 59 *)
TON_1(IN := MarkTableOn AND ((DuctSelected AND MatlAtMarkTable) OR NOT DuctSelected), PT := ReverseDelay);
TableRev3 := TON_1.Q;

(* Network 60: Pusher Output *)
_e23(CLK := MarkPushComplete);
IF TableStyle3 AND _e23.Q THEN PusherOffDelay := DINT_TO_TIME(MarkPStartDelay); END_IF;

(* Network 61 *)
_e24(CLK := MarkPushComplete);
IF TableStyle3 AND _e24.Q THEN MPRTime := DINT_TO_TIME(MarkPStopDelay); END_IF;

(* Network 62 *)
TON_13(IN := MarkPushComplete AND MarkConveyorDelayFwd, PT := MPRTime);
MarkPushReady := TON_13.Q;

(* Network 63 *)
TOF_0(IN := TableFwd3 AND MarkPushReady, PT := PusherOffDelay);
PushValve3 := TOF_0.Q;

(* Network 64: Gate Raise Output *)
_e25(CLK := MarkPusherStop);
IF _e25.Q AND TableStyle3 THEN GateLowerDelay := DINT_TO_TIME(MarkPPauseDwell); END_IF;

(* Network 65 *)
TOF_1(IN := MarkPusherStop, PT := GateLowerDelay);
MarkPusherStopDOB := TOF_1.Q;

(* Network 66 *)
Gate3 := MarkPusherStopDOB OR (MarkTableOn AND NOT DuctSelected);

(* Network 67: Switch local variables to physical outputs based on table type. *)
MarkTableFwd := (TableFwd3 AND TableStyle3) OR (TableFwd2 AND TableStyle2);

(* Network 68 *)
MarkTableRev := (TableRev3 AND TableStyle3) OR (TableRev2 AND TableStyle2);

(* Network 69 *)
MarkPshrFwd := (PushValve3 AND TableStyle3) OR (PushValve2 AND TableStyle2);

(* Network 70 *)
MarkPusherReverse := (TableStyle3 AND MarkTableOn AND NOT MarkPshrFwd AND Mark3PusherHome) OR Psh8 OR MarkTTPusherJogRevPB;

(* Network 71 *)
MarkGateRaise := (Gate3 AND TableStyle3) OR (Gate2 AND TableStyle2);
END_PROGRAM
```

### Program Logical/MarkRF (IEC)

#### Variables.var
```iecst
VAR
	AbsDiff : DINT;
	CheckPosition : BOOL;
	GoodToGo : BOOL;
	Homed : BOOL;
	InPosition : BOOL;
	NotInSlowBand : BOOL;
	RefInProcess : BOOL;
	ResetMarkHoming : BOOL;
	ResetMarkSet : BOOL;
	ReturnTarget : DINT;
	ScaledTarget : DINT;
	Scaler : REAL;
	ScalerRef : DINT;
	SetStepA : BOOL;
	SetStepB : BOOL;
	StepAComplete : BOOL;
	StepBWorking : BOOL;
	TargetOk : BOOL;
	TargetTooSmall : BOOL;
	TempStat : INT;
	TON_0 : TON;
	TON_1 : TON;
	TON_2 : TON;
	TP_0 : TP;
	TP_1 : TP;
	WaitToChange : BOOL;
	RTGTME : BOOL;
	MarkSignaling : BOOL;
	TON_3 : TON;
	SignalTimeUp : BOOL;
	MarkSettingUp : BOOL;
END_VAR
```

#### Cyclic.ld
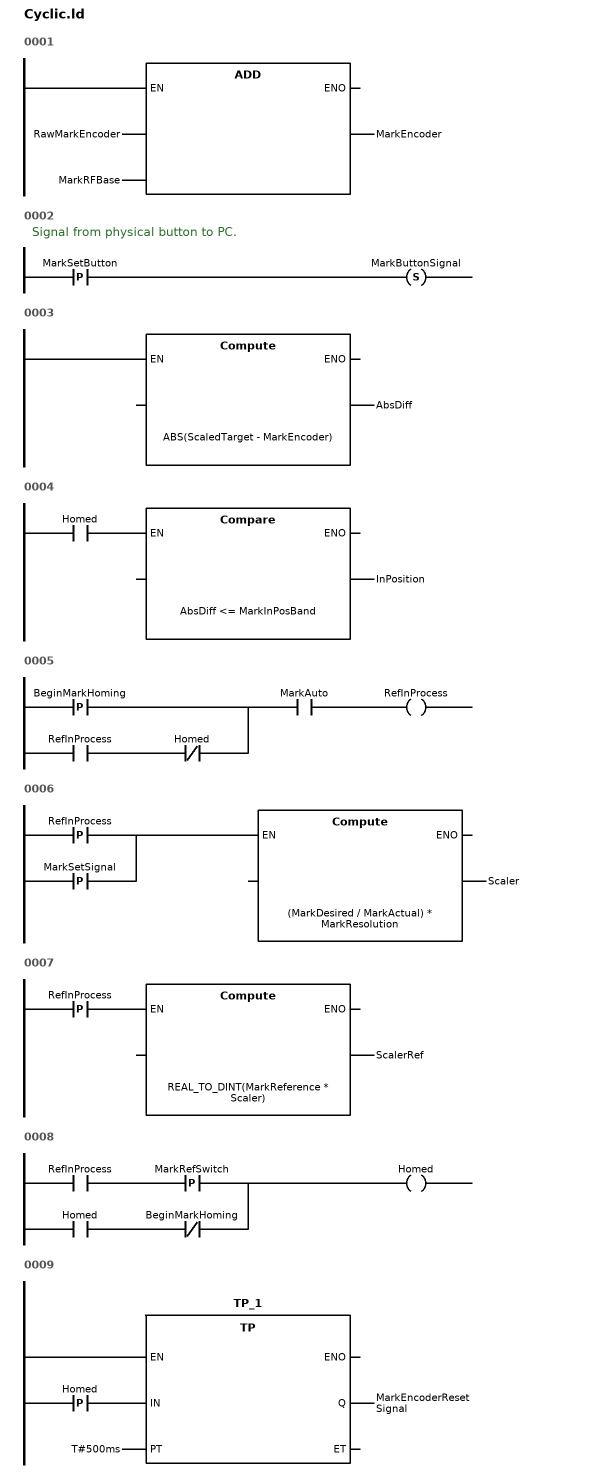
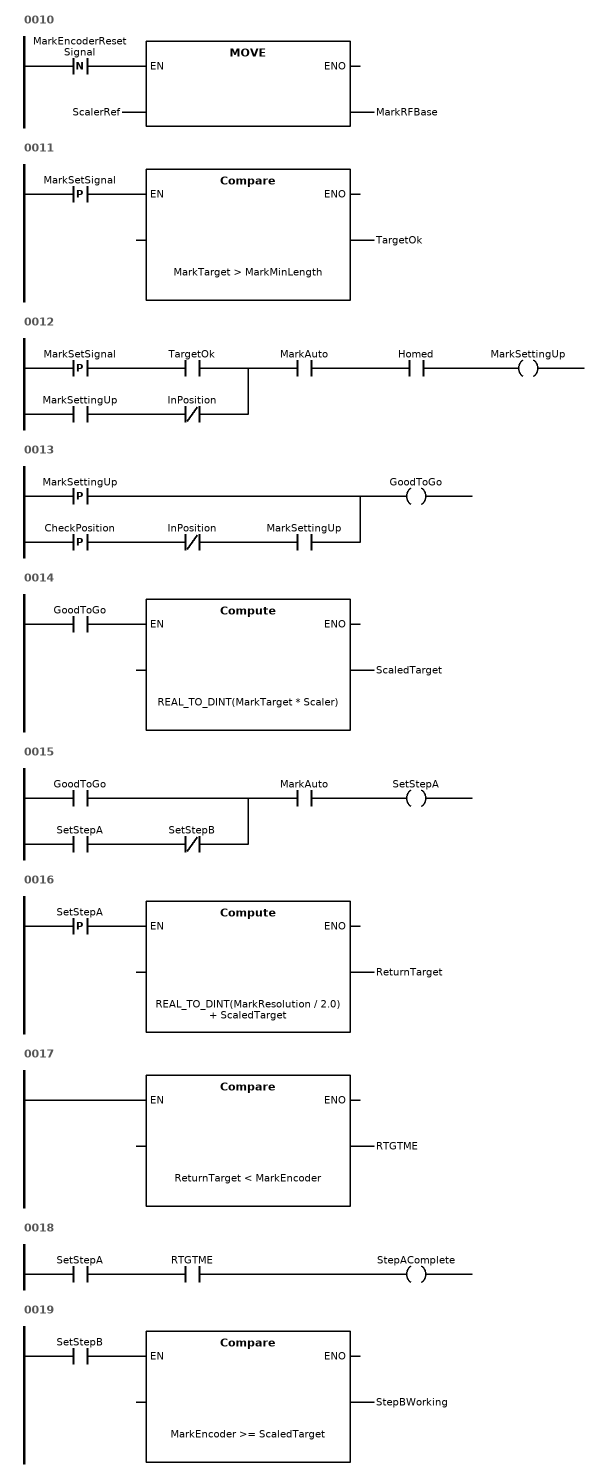
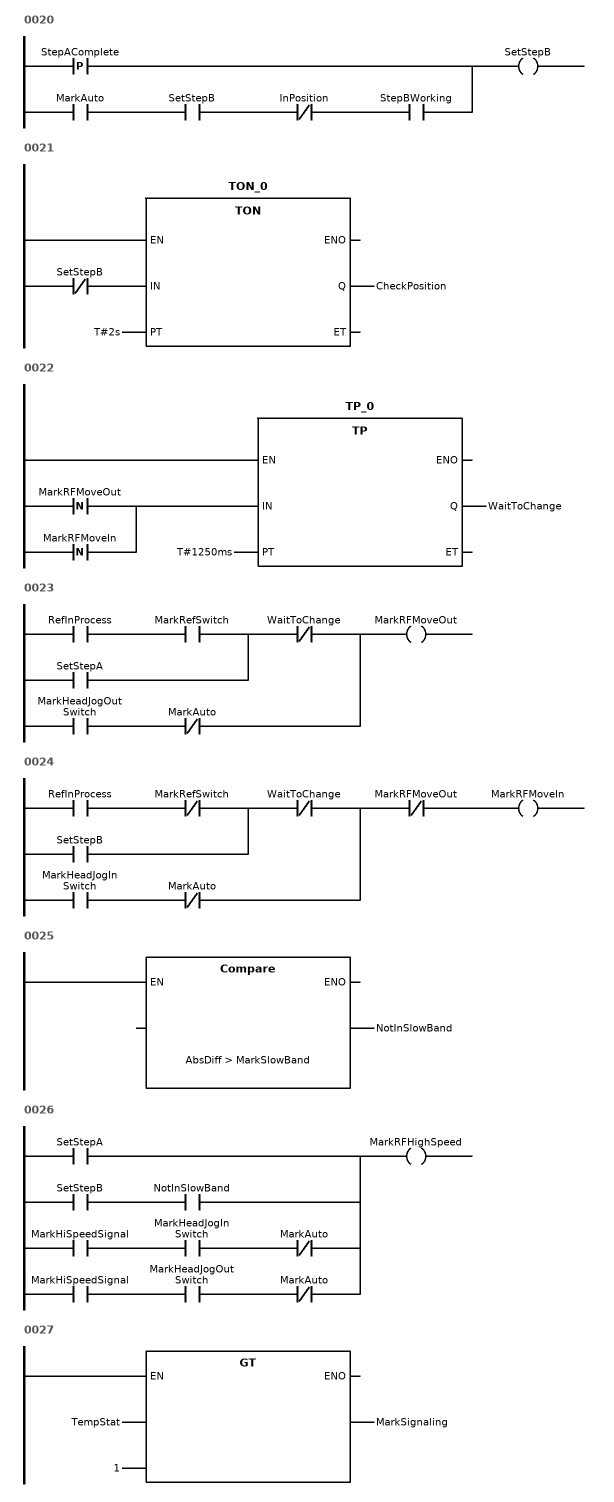
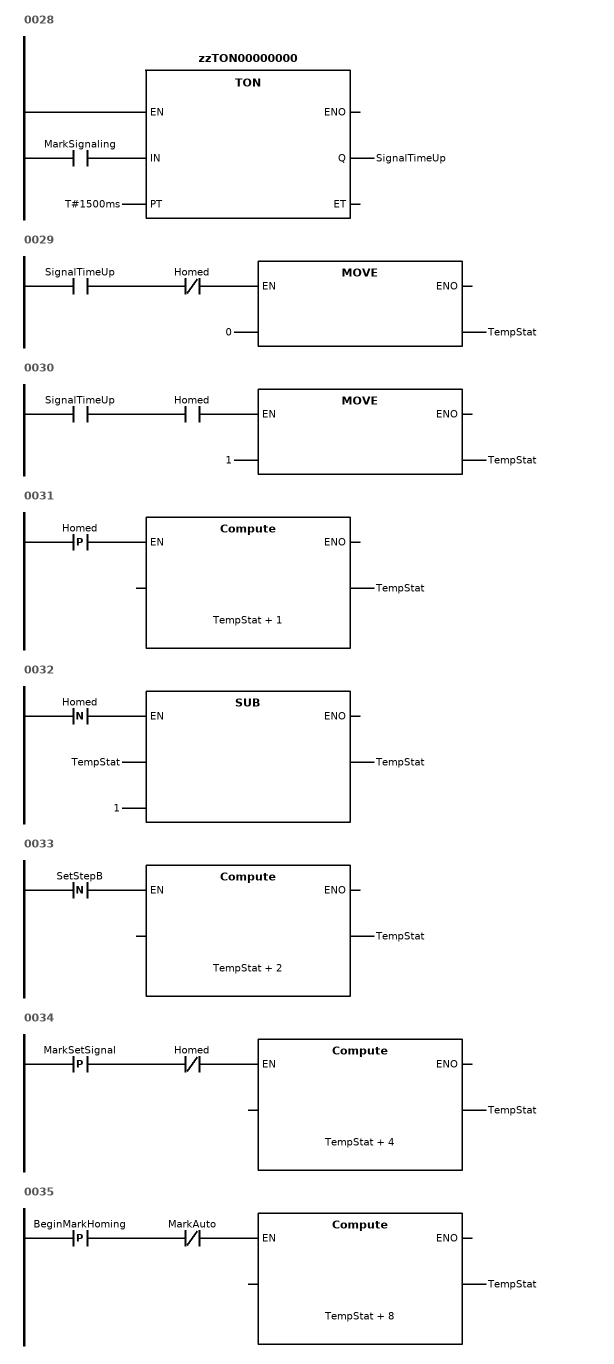
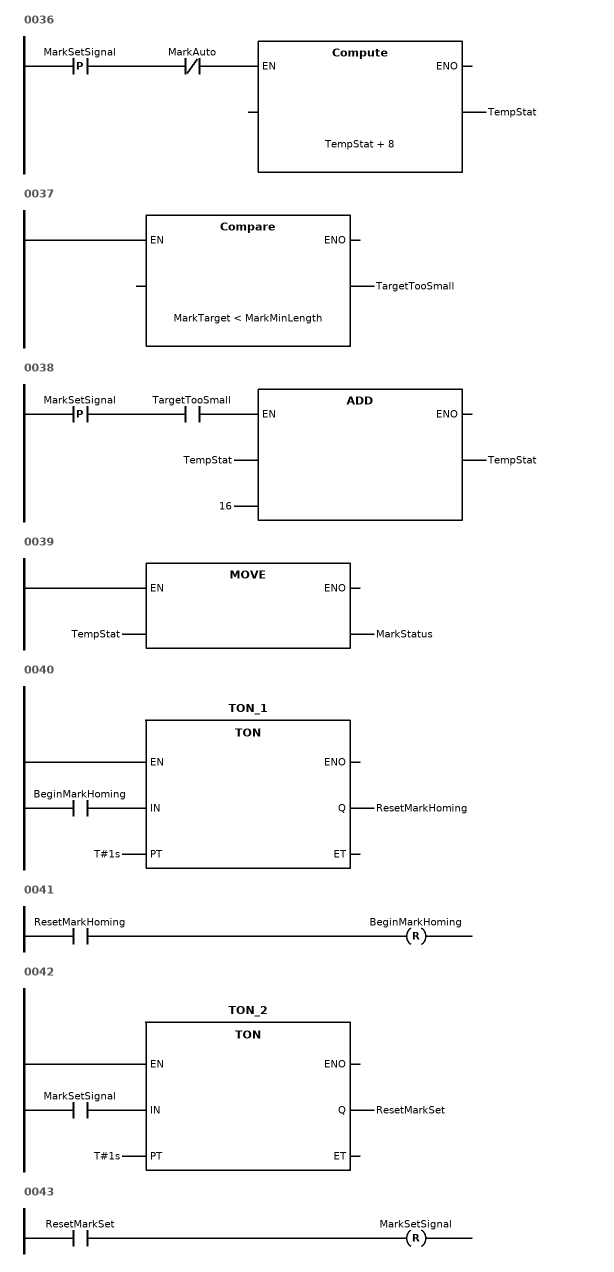
Ladder, written as Structured Text:
```iecst
PROGRAM _CYCLIC
VAR
    _e1 : R_TRIG;
    _e2 : R_TRIG;
    _e3 : R_TRIG;
    _e4 : R_TRIG;
    _e5 : R_TRIG;
    _e6 : R_TRIG;
    _e7 : R_TRIG;
    _e8 : F_TRIG;
    _e9 : R_TRIG;
    _e10 : R_TRIG;
    _e11 : R_TRIG;
    _e12 : R_TRIG;
    _e13 : R_TRIG;
    _e14 : R_TRIG;
    _e15 : F_TRIG;
    _e16 : F_TRIG;
    _e17 : R_TRIG;
    _e18 : F_TRIG;
    _e19 : F_TRIG;
    _e20 : R_TRIG;
    _e21 : R_TRIG;
    _e22 : R_TRIG;
    _e23 : R_TRIG;
END_VAR
(* Network 1 *)
MarkEncoder := RawMarkEncoder + MarkRFBase;

(* Network 2: Signal from physical button to PC. *)
_e1(CLK := MarkSetButton);
IF _e1.Q THEN MarkButtonSignal := TRUE; END_IF;

(* Network 3 *)
AbsDiff := ABS(ScaledTarget - MarkEncoder);

(* Network 4 *)
IF Homed THEN InPosition := AbsDiff <= MarkInPosBand; END_IF;

(* Network 5 *)
_e2(CLK := BeginMarkHoming);
RefInProcess := (_e2.Q OR (RefInProcess AND NOT Homed)) AND MarkAuto;

(* Network 6 *)
_e3(CLK := RefInProcess);
_e4(CLK := MarkSetSignal);
IF _e3.Q OR _e4.Q THEN Scaler := (MarkDesired / MarkActual) * MarkResolution; END_IF;

(* Network 7 *)
_e5(CLK := RefInProcess);
IF _e5.Q THEN ScalerRef := REAL_TO_DINT(MarkReference * Scaler); END_IF;

(* Network 8 *)
_e6(CLK := MarkRefSwitch);
Homed := (RefInProcess AND _e6.Q) OR (Homed AND NOT BeginMarkHoming);

(* Network 9 *)
_e7(CLK := Homed);
TP_1(IN := _e7.Q, PT := T#500ms);
MarkEncoderResetSignal := TP_1.Q;

(* Network 10 *)
_e8(CLK := MarkEncoderResetSignal);
IF _e8.Q THEN MarkRFBase := ScalerRef; END_IF;

(* Network 11 *)
_e9(CLK := MarkSetSignal);
IF _e9.Q THEN TargetOk := MarkTarget > MarkMinLength; END_IF;

(* Network 12 *)
_e10(CLK := MarkSetSignal);
MarkSettingUp := ((_e10.Q AND TargetOk) OR (MarkSettingUp AND NOT InPosition)) AND MarkAuto AND Homed;

(* Network 13 *)
_e11(CLK := MarkSettingUp);
_e12(CLK := CheckPosition);
GoodToGo := _e11.Q OR (_e12.Q AND NOT InPosition AND MarkSettingUp);

(* Network 14 *)
IF GoodToGo THEN ScaledTarget := REAL_TO_DINT(MarkTarget * Scaler); END_IF;

(* Network 15 *)
SetStepA := (GoodToGo OR (SetStepA AND NOT SetStepB)) AND MarkAuto;

(* Network 16 *)
_e13(CLK := SetStepA);
IF _e13.Q THEN ReturnTarget := REAL_TO_DINT(MarkResolution / 2.0) + ScaledTarget; END_IF;

(* Network 17 *)
RTGTME := ReturnTarget < MarkEncoder;

(* Network 18 *)
StepAComplete := SetStepA AND RTGTME;

(* Network 19 *)
IF SetStepB THEN StepBWorking := MarkEncoder >= ScaledTarget; END_IF;

(* Network 20 *)
_e14(CLK := StepAComplete);
SetStepB := _e14.Q OR (MarkAuto AND SetStepB AND NOT InPosition AND StepBWorking);

(* Network 21 *)
TON_0(IN := NOT SetStepB, PT := T#2s);
CheckPosition := TON_0.Q;

(* Network 22 *)
_e15(CLK := MarkRFMoveOut);
_e16(CLK := MarkRFMoveIn);
TP_0(IN := _e15.Q OR _e16.Q, PT := T#1250ms);
WaitToChange := TP_0.Q;

(* Network 23 *)
MarkRFMoveOut := (((RefInProcess AND MarkRefSwitch) OR SetStepA) AND NOT WaitToChange) OR (MarkHeadJogOutSwitch AND NOT MarkAuto);

(* Network 24 *)
MarkRFMoveIn := ((((RefInProcess AND NOT MarkRefSwitch) OR SetStepB) AND NOT WaitToChange) OR (MarkHeadJogInSwitch AND NOT MarkAuto)) AND NOT MarkRFMoveOut;

(* Network 25 *)
NotInSlowBand := AbsDiff > MarkSlowBand;

(* Network 26 *)
MarkRFHighSpeed := SetStepA OR (SetStepB AND NotInSlowBand) OR (MarkHiSpeedSignal AND ((MarkHeadJogInSwitch AND NOT MarkAuto) OR (MarkHeadJogOutSwitch AND NOT MarkAuto)));

(* Network 27 *)
MarkSignaling := TempStat > 1;

(* Network 28 *)
zzTON00000000(IN := MarkSignaling, PT := T#1500ms);
SignalTimeUp := zzTON00000000.Q;

(* Network 29 *)
IF SignalTimeUp AND NOT Homed THEN TempStat := 0; END_IF;

(* Network 30 *)
IF SignalTimeUp AND Homed THEN TempStat := 1; END_IF;

(* Network 31 *)
_e17(CLK := Homed);
IF _e17.Q THEN TempStat := TempStat + 1; END_IF;

(* Network 32 *)
_e18(CLK := Homed);
IF _e18.Q THEN TempStat := TempStat - 1; END_IF;

(* Network 33 *)
_e19(CLK := SetStepB);
IF _e19.Q THEN TempStat := TempStat + 2; END_IF;

(* Network 34 *)
_e20(CLK := MarkSetSignal);
IF _e20.Q AND NOT Homed THEN TempStat := TempStat + 4; END_IF;

(* Network 35 *)
_e21(CLK := BeginMarkHoming);
IF _e21.Q AND NOT MarkAuto THEN TempStat := TempStat + 8; END_IF;

(* Network 36 *)
_e22(CLK := MarkSetSignal);
IF _e22.Q AND NOT MarkAuto THEN TempStat := TempStat + 8; END_IF;

(* Network 37 *)
TargetTooSmall := MarkTarget < MarkMinLength;

(* Network 38 *)
_e23(CLK := MarkSetSignal);
IF _e23.Q AND TargetTooSmall THEN TempStat := TempStat + 16; END_IF;

(* Network 39 *)
MarkStatus := TempStat;

(* Network 40 *)
TON_1(IN := BeginMarkHoming, PT := T#1s);
ResetMarkHoming := TON_1.Q;

(* Network 41 *)
IF ResetMarkHoming THEN BeginMarkHoming := FALSE; END_IF;

(* Network 42 *)
TON_2(IN := MarkSetSignal, PT := T#1s);
ResetMarkSet := TON_2.Q;

(* Network 43 *)
IF ResetMarkSet THEN MarkSetSignal := FALSE; END_IF;
END_PROGRAM
```

#### Init.ld
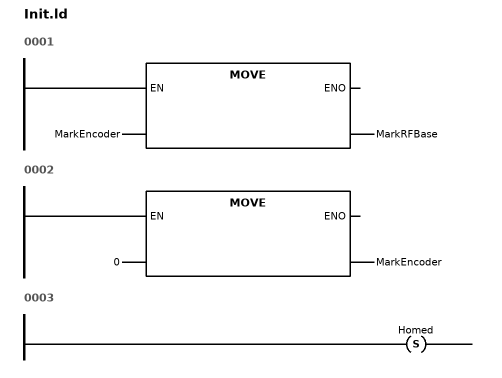
Ladder, written as Structured Text:
```iecst
PROGRAM _INIT
(* Network 1 *)
MarkRFBase := MarkEncoder;

(* Network 2 *)
MarkEncoder := 0;

(* Network 3 *)
Homed := TRUE;
END_PROGRAM
```

### Program Logical/TDCRFPshrs (IEC)

#### Variables.var
```iecst
VAR
	TDCPusherUnlatch : BOOL;
	TDCRFStartPush : BOOL;
	TDCRFP1 : BOOL;
	TDCRFP3 : BOOL;
	TDCPushDelayDone : BOOL;
	TDCRFP2 : BOOL;
	TDCRFP4 : BOOL;
	TDCRFP5 : BOOL;
	TDCRFPTime : TIME;
	TON_0 : TON;
END_VAR
```

#### Cyclic.ld
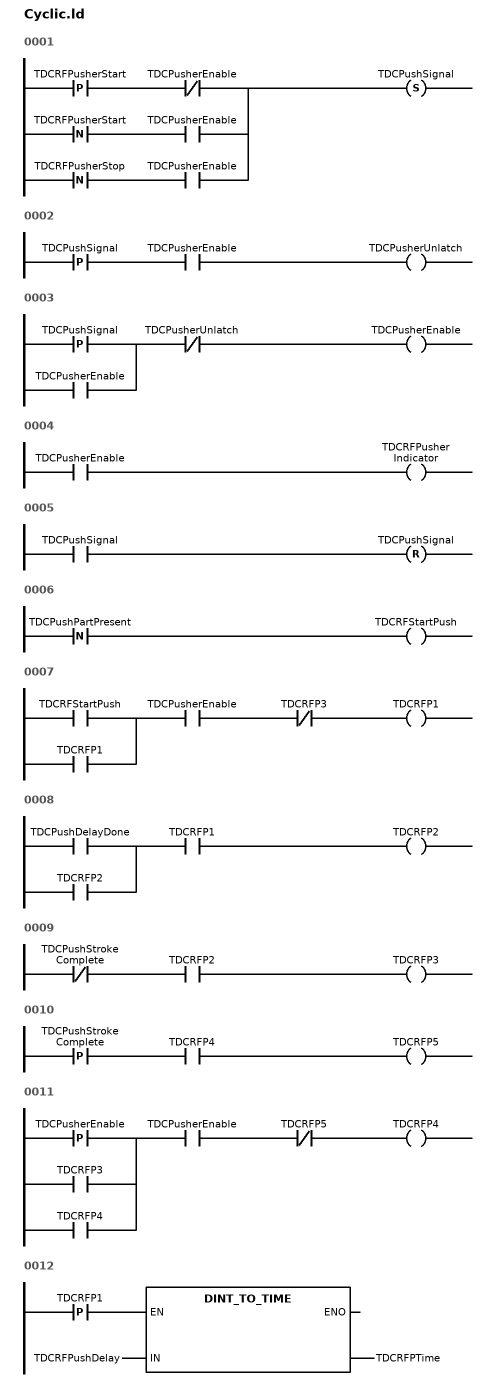
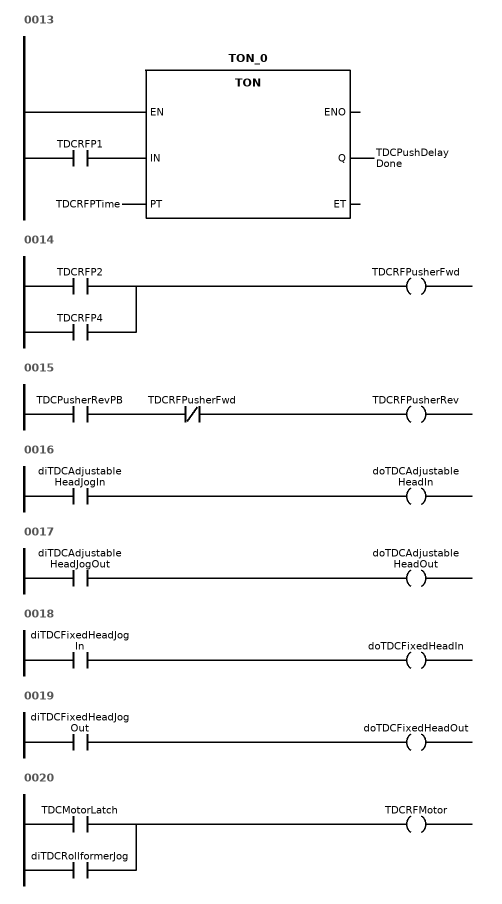
Ladder, written as Structured Text:
```iecst
PROGRAM _CYCLIC
VAR
    _e1 : R_TRIG;
    _e2 : F_TRIG;
    _e3 : F_TRIG;
    _e4 : R_TRIG;
    _e5 : R_TRIG;
    _e6 : F_TRIG;
    _e7 : R_TRIG;
    _e8 : R_TRIG;
    _e9 : R_TRIG;
END_VAR
(* Network 1 *)
_e1(CLK := TDCRFPusherStart);
_e2(CLK := TDCRFPusherStart);
_e3(CLK := TDCRFPusherStop);
IF (_e1.Q AND NOT TDCPusherEnable) OR (_e2.Q AND TDCPusherEnable) OR (_e3.Q AND TDCPusherEnable) THEN
    TDCPushSignal := TRUE;
END_IF;

(* Network 2 *)
_e4(CLK := TDCPushSignal);
TDCPusherUnlatch := _e4.Q AND TDCPusherEnable;

(* Network 3 *)
_e5(CLK := TDCPushSignal);
TDCPusherEnable := (_e5.Q OR TDCPusherEnable) AND NOT TDCPusherUnlatch;

(* Network 4 *)
TDCRFPusherIndicator := TDCPusherEnable;

(* Network 5 *)
IF TDCPushSignal THEN TDCPushSignal := FALSE; END_IF;

(* Network 6 *)
_e6(CLK := TDCPushPartPresent);
TDCRFStartPush := _e6.Q;

(* Network 7 *)
TDCRFP1 := (TDCRFStartPush OR TDCRFP1) AND TDCPusherEnable AND NOT TDCRFP3;

(* Network 8 *)
TDCRFP2 := (TDCPushDelayDone OR TDCRFP2) AND TDCRFP1;

(* Network 9 *)
TDCRFP3 := NOT TDCPushStrokeComplete AND TDCRFP2;

(* Network 10 *)
_e7(CLK := TDCPushStrokeComplete);
TDCRFP5 := _e7.Q AND TDCRFP4;

(* Network 11 *)
_e8(CLK := TDCPusherEnable);
TDCRFP4 := (_e8.Q OR TDCRFP3 OR TDCRFP4) AND TDCPusherEnable AND NOT TDCRFP5;

(* Network 12 *)
_e9(CLK := TDCRFP1);
IF _e9.Q THEN TDCRFPTime := DINT_TO_TIME(TDCRFPushDelay); END_IF;

(* Network 13 *)
TON_0(IN := TDCRFP1, PT := TDCRFPTime);
TDCPushDelayDone := TON_0.Q;

(* Network 14 *)
TDCRFPusherFwd := TDCRFP2 OR TDCRFP4;

(* Network 15 *)
TDCRFPusherRev := TDCPusherRevPB AND NOT TDCRFPusherFwd;

(* Network 16 *)
doTDCAdjustableHeadIn := diTDCAdjustableHeadJogIn;

(* Network 17 *)
doTDCAdjustableHeadOut := diTDCAdjustableHeadJogOut;

(* Network 18 *)
doTDCFixedHeadIn := diTDCFixedHeadJogIn;

(* Network 19 *)
doTDCFixedHeadOut := diTDCFixedHeadJogOut;

(* Network 20 *)
TDCRFMotor := TDCMotorLatch OR diTDCRollformerJog;
END_PROGRAM
```

### Program Logical/GlueApp (IEC)

#### Variables.var
```iecst
VAR
	ApplicatorTypeIs1 : BOOL;
	GlueSprayEnable1 : BOOL;
	ApplicatorTypeIs2 : BOOL;
	LeadDelay : TIME;
	TrailDelay : TIME;
	TON_0 : TON;
	TP_0 : TP;
	StartGlue : BOOL;
	ContinueGlue : BOOL;
	ApplicatorTypeIs3 : BOOL;
	MT0 : BOOL;
	TON_1 : TON;
	MTStartGlue : BOOL;
	MT1 : BOOL;
	MT2 : BOOL;
	MTStopGlue : BOOL;
	ResetMTSequence : BOOL;
	CCLength : TIME;
	TP_1 : TP;
	TP_2 : TP;
	TP_3 : TP;
	FTRSDelay : BOOL;
	FTRTime : TIME;
	Clean1 : BOOL;
	TON_2 : TON;
	C1Done : BOOL;
	Clean2 : BOOL;
	TON_3 : TON;
	C2Done : BOOL;
	Clean3 : BOOL;
	GFPB1 : BOOL;
	GFPB2 : BOOL;
	TON_4 : TON;
	GFPBTmr : BOOL;
	GFPBReset : BOOL;
	TON_5 : TON;
END_VAR
```

#### Cyclic.ld
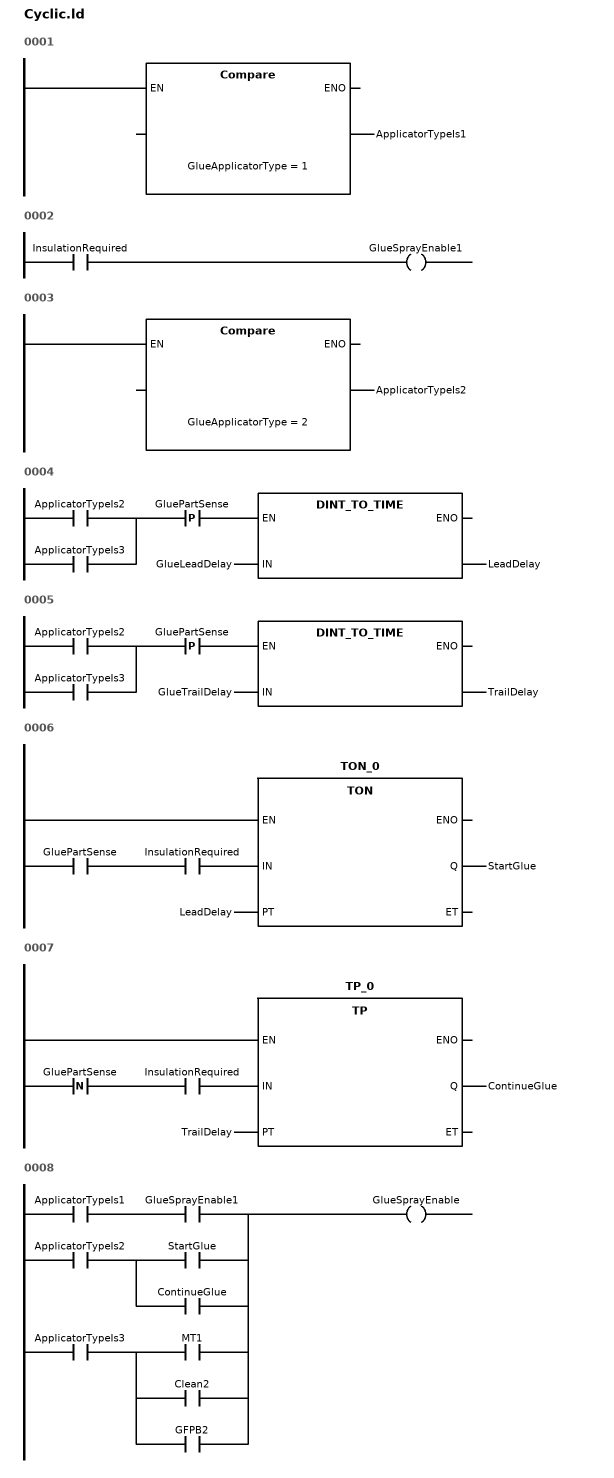
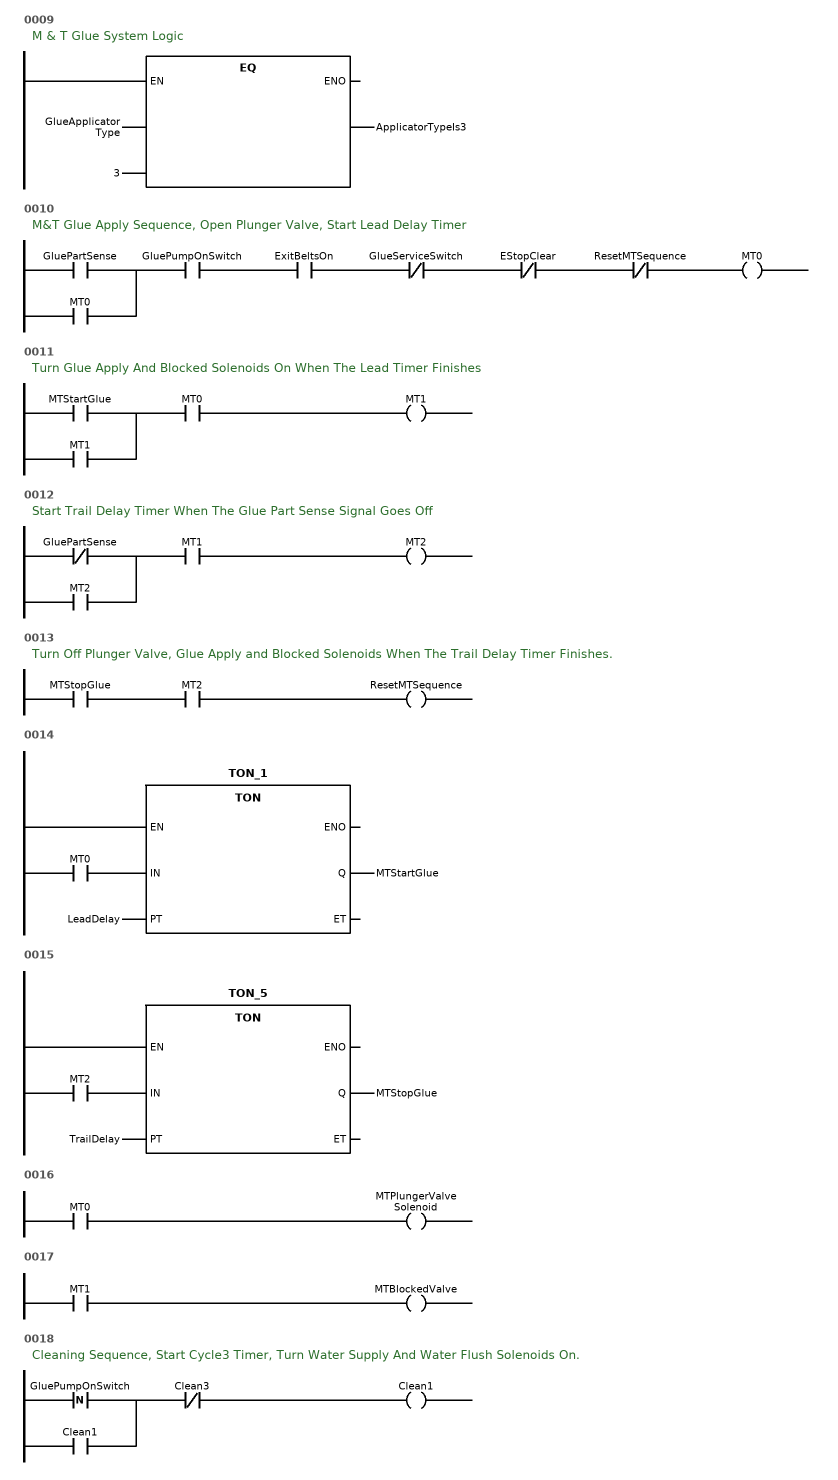
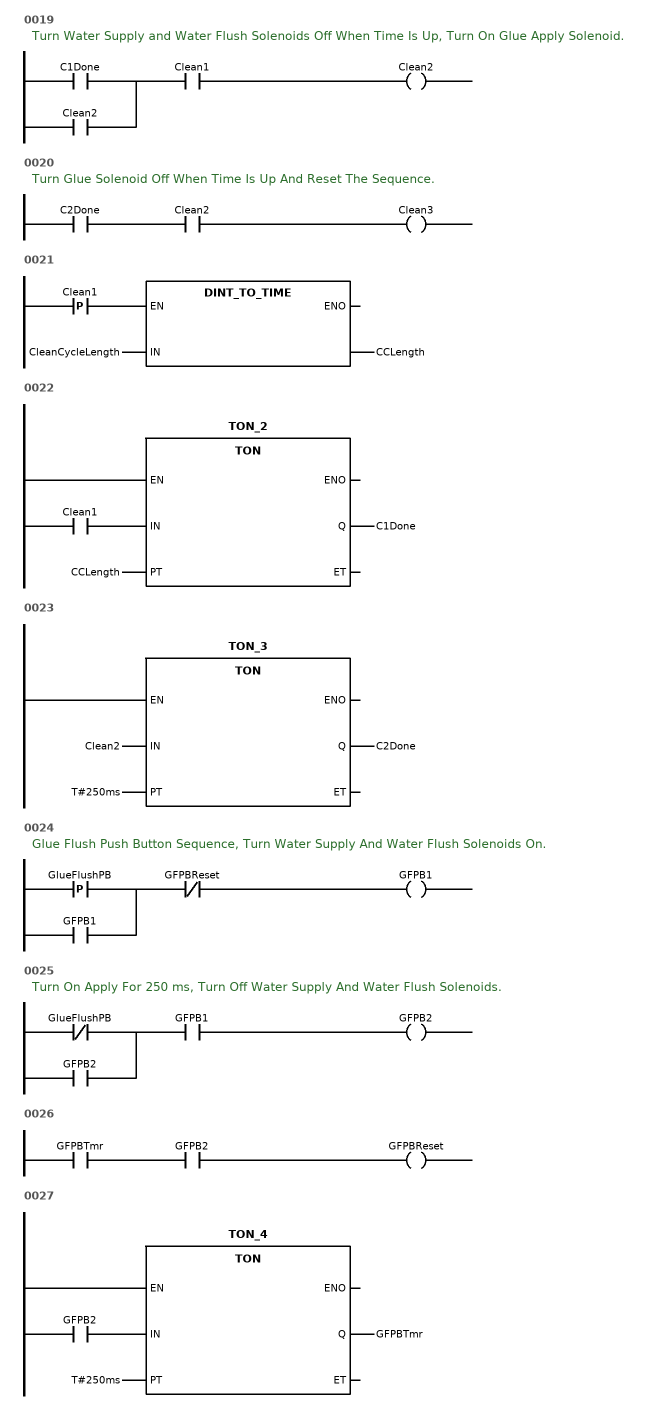
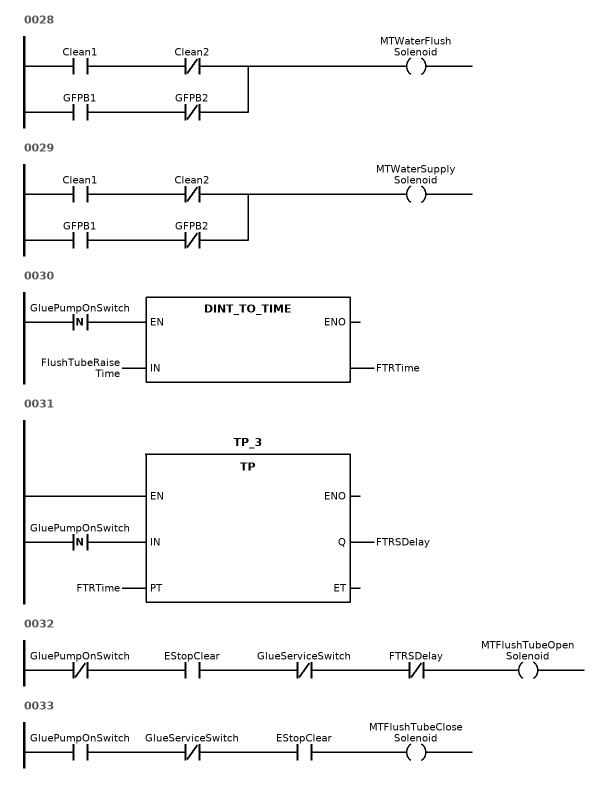
Ladder, written as Structured Text:
```iecst
PROGRAM _CYCLIC
VAR
    _e1 : R_TRIG;
    _e2 : R_TRIG;
    _e3 : F_TRIG;
    _e4 : F_TRIG;
    _e5 : R_TRIG;
    _e6 : R_TRIG;
    _e7 : F_TRIG;
    _e8 : F_TRIG;
END_VAR
(* Network 1 *)
ApplicatorTypeIs1 := GlueApplicatorType = 1;

(* Network 2 *)
GlueSprayEnable1 := InsulationRequired;

(* Network 3 *)
ApplicatorTypeIs2 := GlueApplicatorType = 2;

(* Network 4 *)
_e1(CLK := GluePartSense);
IF (ApplicatorTypeIs2 OR ApplicatorTypeIs3) AND _e1.Q THEN
    LeadDelay := DINT_TO_TIME(GlueLeadDelay);
END_IF;

(* Network 5 *)
_e2(CLK := GluePartSense);
IF (ApplicatorTypeIs2 OR ApplicatorTypeIs3) AND _e2.Q THEN
    TrailDelay := DINT_TO_TIME(GlueTrailDelay);
END_IF;

(* Network 6 *)
TON_0(IN := GluePartSense AND InsulationRequired, PT := LeadDelay);
StartGlue := TON_0.Q;

(* Network 7 *)
_e3(CLK := GluePartSense);
TP_0(IN := _e3.Q AND InsulationRequired, PT := TrailDelay);
ContinueGlue := TP_0.Q;

(* Network 8 *)
GlueSprayEnable := (ApplicatorTypeIs1 AND GlueSprayEnable1) OR (ApplicatorTypeIs2 AND (StartGlue OR ContinueGlue)) OR (ApplicatorTypeIs3 AND (MT1 OR Clean2 OR GFPB2));

(* Network 9: M & T Glue System Logic *)
ApplicatorTypeIs3 := GlueApplicatorType = 3;

(* Network 10: M&T Glue Apply Sequence, Open Plunger Valve, Start Lead Delay Timer *)
MT0 := (GluePartSense OR MT0) AND GluePumpOnSwitch AND ExitBeltsOn AND NOT GlueServiceSwitch AND NOT EStopClear AND NOT ResetMTSequence;

(* Network 11: Turn Glue Apply And Blocked Solenoids On When The Lead Timer Finishes *)
MT1 := (MTStartGlue OR MT1) AND MT0;

(* Network 12: Start Trail Delay Timer When The Glue Part Sense Signal Goes Off *)
MT2 := (NOT GluePartSense OR MT2) AND MT1;

(* Network 13: Turn Off Plunger Valve, Glue Apply and Blocked Solenoids When The Trail Delay Timer Finishes. *)
ResetMTSequence := MTStopGlue AND MT2;

(* Network 14 *)
TON_1(IN := MT0, PT := LeadDelay);
MTStartGlue := TON_1.Q;

(* Network 15 *)
TON_5(IN := MT2, PT := TrailDelay);
MTStopGlue := TON_5.Q;

(* Network 16 *)
MTPlungerValveSolenoid := MT0;

(* Network 17 *)
MTBlockedValve := MT1;

(* Network 18: Cleaning Sequence, Start Cycle3 Timer, Turn Water Supply And Water Flush Solenoids On. *)
_e4(CLK := GluePumpOnSwitch);
Clean1 := (_e4.Q OR Clean1) AND NOT Clean3;

(* Network 19: Turn Water Supply and Water Flush Solenoids Off When Time Is Up, Turn On Glue Apply Solenoid. *)
Clean2 := (C1Done OR Clean2) AND Clean1;

(* Network 20: Turn Glue Solenoid Off When Time Is Up And Reset The Sequence. *)
Clean3 := C2Done AND Clean2;

(* Network 21 *)
_e5(CLK := Clean1);
IF _e5.Q THEN CCLength := DINT_TO_TIME(CleanCycleLength); END_IF;

(* Network 22 *)
TON_2(IN := Clean1, PT := CCLength);
C1Done := TON_2.Q;

(* Network 23 *)
TON_3(IN := Clean2, PT := T#250ms);
C2Done := TON_3.Q;

(* Network 24: Glue Flush Push Button Sequence, Turn Water Supply And Water Flush Solenoids On. *)
_e6(CLK := GlueFlushPB);
GFPB1 := (_e6.Q OR GFPB1) AND NOT GFPBReset;

(* Network 25: Turn On Apply For 250 ms, Turn Off Water Supply And Water Flush Solenoids. *)
GFPB2 := (NOT GlueFlushPB OR GFPB2) AND GFPB1;

(* Network 26 *)
GFPBReset := GFPBTmr AND GFPB2;

(* Network 27 *)
TON_4(IN := GFPB2, PT := T#250ms);
GFPBTmr := TON_4.Q;

(* Network 28 *)
MTWaterFlushSolenoid := (Clean1 AND NOT Clean2) OR (GFPB1 AND NOT GFPB2);

(* Network 29 *)
MTWaterSupplySolenoid := (Clean1 AND NOT Clean2) OR (GFPB1 AND NOT GFPB2);

(* Network 30 *)
_e7(CLK := GluePumpOnSwitch);
IF _e7.Q THEN FTRTime := DINT_TO_TIME(FlushTubeRaiseTime); END_IF;

(* Network 31 *)
_e8(CLK := GluePumpOnSwitch);
TP_3(IN := _e8.Q, PT := FTRTime);
FTRSDelay := TP_3.Q;

(* Network 32 *)
MTFlushTubeOpenSolenoid := NOT GluePumpOnSwitch AND EStopClear AND NOT GlueServiceSwitch AND NOT FTRSDelay;

(* Network 33 *)
MTFlushTubeCloseSolenoid := GluePumpOnSwitch AND NOT GlueServiceSwitch AND EStopClear;
END_PROGRAM
```

### Program Logical/Insulmatic (IEC)

#### Variables.var
```iecst
VAR
	T13 : TIME;
	SP2 : BOOL;
	TP_0 : TP;
	SP1 : BOOL;
	TON_0 : TON;
	BTimer2Done : BOOL;
	B0 : BOOL;
	B1 : BOOL;
	BTimer1Done : BOOL;
	B2 : BOOL;
	T9 : TIME;
	T6 : TIME;
	TON_1 : TON;
	TON_2 : TON;
	FRTimer2Done : BOOL;
	FR0 : BOOL;
	FR1 : BOOL;
	FRTimer1Done : BOOL;
	FR2 : BOOL;
	TempFRDelay : DINT;
	T4 : TIME;
	T2 : TIME;
	TempFR2Delay : DINT;
	TON_3 : TON;
	TON_4 : TON;
	PRTimer2Done : BOOL;
	PR0 : BOOL;
	PR1 : BOOL;
	PRTimer1Done : BOOL;
	PR2 : BOOL;
	T7 : TIME;
	T3 : TIME;
	TON_5 : TON;
	TON_6 : TON;
	HLTimer2Done : BOOL;
	HLwSq0 : BOOL;
	HLwSq1 : BOOL;
	HLwoSq0 : BOOL;
	HLwoSq1 : BOOL;
	HLTimer1Done : BOOL;
	HLwoSq2 : BOOL;
	HLTempTimer : DINT;
	T5 : TIME;
	TON_7 : TON;
	T8 : TIME;
	TON_8 : TON;
	SwingBlade : BOOL;
	SwingCount : DINT;
	SwingRem : DINT;
	SCIsBig : BOOL;
	SwingCountIsEven : BOOL;
END_VAR
```
